# B&R Automation Studio project SortingStation
Automation Studio 4.12.4.107 SP; technology packages: mapp 5.23.1, mappCockpit 5.23.0, mappMotion 5.23.1, mappView 5.23.0

## Configuration Configuration

CPU X20CP1686X, AutomationRuntime H4.93, Build 4.1.2, Vc V4.73.0

### Task classes (Cpu.sw)
```
Cyclic#1:
  RSModelSor <- RSModelSort.prg
  ConveyorPr <- Source.Conveyor.ConveyorProgram.prg
  PuncherPro <- Source.Puncher.PuncherProgram.prg
Cyclic#2 (cycle 12000 us, tolerance 12000 us):
  MainMachin <- Source.MainMachine.MainMachineProgram.prg
  ColourSort <- Source.ColourSorter.ColourSorterProgram.prg
Cyclic#4:
  RecipesPro <- Source.Infrastructure.Recipes.RecipesProgram.prg
  Alarms <- Source.Infrastructure.Alarms.Alarms.prg
  HMIProgram <- Source.HMI.HMIProgram.prg
DataObjects: McAcpSys
NcDataObjects: McDriveLog
Binaries: TCLang, McAcpDrv, udbdef, McAcpSim, mvLoader, arflatprv, mCoWebSc, TCData, FWRules, arcoal, arsvcreg, OpcUaSrv, Settings, iomap, asfw, Role, ashwac, sysconf, AxisConfig, arconfig, AlarmsCore, AlarmsHist, TC, ashwd, User, Cam, Users
Libraries: McBase, MpAxis, McAxis, MpBase, McAcpAx, CoTrace, AsZip, FileIO, runtime, MpAlarmX, astime, standard, asstring, MpServer, MpFile, MpUserX, MpRecipe, sys_lib, asieccon, asbrstr, dataobj, asepl, asusb, aruser, arssl, powerlnk, arcert, ashw, aseth
```

### Hardware
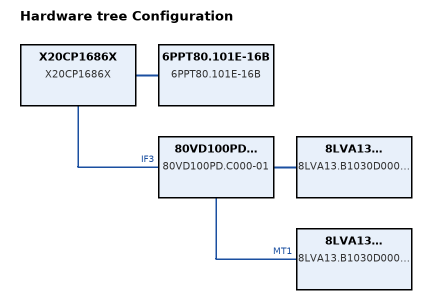
```
6PPT80.101E-16B : 6PPT80.101E-16B v1.0.6.0  [ETH1 -> X20CP1686X.IF2 [Cable Type=PowerlinkCable, Length=10, Version=1.0.0.3]]
  Terminal = true
  Startmode = 2
  Mode = Manual
  InternetAddress = 192.168.0.4
  Subnetmask = 255.255.255.0
  ScreenRotation = 180
  PasswordVNC = 
  SelectedFavoriteWeb = 192.168.0.3:81
  BrowserVKeyboard = 0
  PasswordCIFS = 
  PasswordService = 
80VD100PD.C000-01 : 80VD100PD.C000-01 v2.5.0.0  [PLK1 -> X20CP1686X.IF3 (NodeNumber=1) [Cable Type=PowerlinkCable, Length=10, Version=1.0.0.3]; MT2 -> 8LVA13.B1030D000-0.MT]
  DriveConfiguration/Module:
    McAcoposTypeID = AcoposMicroDConfig
    ActivateACOPOSSimulationOnPLC = 1
  DriveConfiguration/Channel[1]/RealAxis:
    AxisReference = gAxisConveyorMpLink
    MechanicalElementsIsInvisible = 0
  DriveConfiguration/Channel[1]/RealAxis/MechanicalElements/Gearbox:
    InputIsReadOnly = 0
    Input = 1
    OutputIsReadOnly = 0
    Output = 1
  DriveConfiguration/Channel[1]/RealAxis/MechanicalElements/RotaryToLinearTransformation:
    ReferenceDistanceIsReadOnly = 0
    ReferenceDistance = 1
  DriveConfiguration/Channel[1]/RealAxis/Controller:
    ModeIsReadOnly = 0
    Mode = PositionController
  DriveConfiguration/Channel[1]/RealAxis/Controller/Mode/Position:
    ProportionalGain = 50.0
    IntegrationTime = 0.0
    PredictionTime = 0.0004
    TotalDelayTime = 0.0004
  DriveConfiguration/Channel[1]/RealAxis/Controller/Mode/Speed:
    ProportionalGainIsReadOnly = 0
    ProportionalGain = 2.0
    IntegrationTimeIsReadOnly = 0
    IntegrationTime = 0.0
    FilterTimeIsReadOnly = 0
    FilterTime = 0.0
  DriveConfiguration/Channel[1]/RealAxis/Controller/Mode/LoopFilters:
    LoopFilterXIsReadOnly = 0
    LoopFilter1 = NotUsed
    LoopFilter2 = NotUsed
    LoopFilter3 = NotUsed
  DriveConfiguration/Channel[1]/RealAxis/Homing:
    ModeIsReadOnly = 0
    Mode = Direct
  DriveConfiguration/Channel[1]/RealAxis/Homing/Mode:
    Position = 0.0
    ReferencePulse = NotUsed
  DriveConfiguration/Channel[1]/RealAxis/Homing:
    RestorePositionVariable = 
  DriveConfiguration/Channel[1]/RealAxis/StopReaction:
    QuickstopIsReadOnly = 0
    Quickstop = DecelerationLimit
    DriveErrorIsReadOnly = 0
    DriveError = DecelerationLimit
  DriveConfiguration/Channel[1]/RealAxis/MovementErrorLimits:
    PositionError = 1.0
    VelocityErrorMonitoring = Automatic1
  DriveConfiguration/Channel[1]/RealAxis:
    JerkFilterIsReadOnly = 0
    JerkFilter = NotUsed
    ZeroVibrationFilter = NotUsed
  DriveConfiguration/Channel[1]/RealAxis/DigitalInputs/HomingSwitch:
    SourceIsReadOnly = 0
    Source = NotUsed
    Level = High
  DriveConfiguration/Channel[1]/RealAxis/DigitalInputs/PositiveLimitSwitch:
    SourceIsReadOnly = 0
    Source = NotUsed
    Level = High
  DriveConfiguration/Channel[1]/RealAxis/DigitalInputs/NegativeLimitSwitch:
    SourceIsReadOnly = 0
    Source = NotUsed
    Level = High
  DriveConfiguration/Channel[1]/RealAxis/DigitalInputs/Trigger1:
    Source = X2Trigger1
    Level = High
  DriveConfiguration/Channel[1]/RealAxis/DigitalInputs/Trigger2:
    Source = X2Trigger2
    Level = High
  DriveConfiguration/Channel[1]/RealAxis/DigitalInputs/Quickstop:
    Input = NotUsed
  DriveConfiguration/Channel[1]/RealAxis/Simulation:
    SimulationModeOnPLC = SetValueGeneration
    SimulationModeOnACOPOS = NotUsed
  DriveConfiguration/Channel[2]/RealAxis:
    AxisReference = gAxisPuncherMpLink
    MechanicalElementsIsInvisible = 0
  DriveConfiguration/Channel[2]/RealAxis/MechanicalElements/Gearbox:
    InputIsReadOnly = 0
    Input = 1
    OutputIsReadOnly = 0
    Output = 1
  DriveConfiguration/Channel[2]/RealAxis/MechanicalElements/RotaryToLinearTransformation:
    ReferenceDistanceIsReadOnly = 0
    ReferenceDistance = 1
  DriveConfiguration/Channel[2]/RealAxis/Controller:
    ModeIsReadOnly = 0
    Mode = PositionController
  DriveConfiguration/Channel[2]/RealAxis/Controller/Mode/Position:
    ProportionalGain = 50.0
    IntegrationTime = 0.0
    PredictionTime = 0.0004
    TotalDelayTime = 0.0004
  DriveConfiguration/Channel[2]/RealAxis/Controller/Mode/Speed:
    ProportionalGainIsReadOnly = 0
    ProportionalGain = 2.0
    IntegrationTimeIsReadOnly = 0
    IntegrationTime = 0.0
    FilterTimeIsReadOnly = 0
    FilterTime = 0.0
  DriveConfiguration/Channel[2]/RealAxis/Controller/Mode/LoopFilters:
    LoopFilterXIsReadOnly = 0
    LoopFilter1 = NotUsed
    LoopFilter2 = NotUsed
    LoopFilter3 = NotUsed
  DriveConfiguration/Channel[2]/RealAxis/Homing:
    ModeIsReadOnly = 0
    Mode = Direct
  DriveConfiguration/Channel[2]/RealAxis/Homing/Mode:
    Position = 0.0
    ReferencePulse = NotUsed
  DriveConfiguration/Channel[2]/RealAxis/Homing:
    RestorePositionVariable = 
  DriveConfiguration/Channel[2]/RealAxis/StopReaction:
    QuickstopIsReadOnly = 0
    Quickstop = DecelerationLimit
    DriveErrorIsReadOnly = 0
    DriveError = DecelerationLimit
  DriveConfiguration/Channel[2]/RealAxis/MovementErrorLimits:
    PositionError = 1.0
    VelocityErrorMonitoring = Automatic1
  DriveConfiguration/Channel[2]/RealAxis:
    JerkFilterIsReadOnly = 0
    JerkFilter = NotUsed
    ZeroVibrationFilter = NotUsed
  DriveConfiguration/Channel[2]/RealAxis/DigitalInputs/HomingSwitch:
    SourceIsReadOnly = 0
    Source = NotUsed
    Level = High
  DriveConfiguration/Channel[2]/RealAxis/DigitalInputs/PositiveLimitSwitch:
    SourceIsReadOnly = 0
    Source = NotUsed
    Level = High
  DriveConfiguration/Channel[2]/RealAxis/DigitalInputs/NegativeLimitSwitch:
    SourceIsReadOnly = 0
    Source = NotUsed
    Level = High
  DriveConfiguration/Channel[2]/RealAxis/DigitalInputs/Trigger1:
    Source = X2Trigger1
    Level = High
  DriveConfiguration/Channel[2]/RealAxis/DigitalInputs/Trigger2:
    Source = X2Trigger2
    Level = High
  DriveConfiguration/Channel[2]/RealAxis/DigitalInputs/Quickstop:
    Input = NotUsed
  DriveConfiguration/Channel[2]/RealAxis/Simulation:
    SimulationModeOnPLC = SetValueGeneration
    SimulationModeOnACOPOS = NotUsed
  DriveConfiguration/Channel[2]/RealAxis/AxisFeatures:
    FeatureRef[1] = CamAutomat
8LVA13.B1030D000-0 : 8LVA13.B1030D000-0 v2.2.0.3  [MT -> 80VD100PD.C000-01.MT2]
  M1/MotorParameters:
    MOTOR_AMB_TEMP_RATED = 40
8LVA13.B1030D000-0a : 8LVA13.B1030D000-0 v2.2.0.3  [MT -> 80VD100PD.C000-01.MT1]
  M1/MotorParameters:
    MOTOR_AMB_TEMP_RATED = 40
X20CP1686X : X20CP1686X v1.8.0.0
  Connector IF2:
    ActivateDevice = 1
    Mode = Manual
    InternetAddress = 192.168.0.3
    SubnetMask = 255.255.255.0
    ActivateSnmp = 2
  ConfigurationID = SortingStation_Configuration
  VolatileGlobalPvSize = 125535
  TimerDeviceType = EPLX2X
  TimerDevice = X20CP1686X.IF3
  Cyclic1Tolerance = 0
  Cyclic2Duration = 12000
  Cyclic2Tolerance = 12000
  FileDevice1
  FileDeviceName1 = RECIPES
  FileDevicePath1 = USER_PATH\recipes
  FtpUser1
  FtpUsername1 = admin
  FtpUserPassword1 = hWQDzdDXjPZQ9N0GtnGX4GsrlK/JakopLOxsvgAIz6U=
  FtpUserSalt1 = DV/Yji4l
  FTPAccessRight1 = 0
  FTPdevice1 = ALL
  ActivateOpcUa = 1
  OpcUaInformationModels_PV_Version = 2
  OpcUaInformationModel_Facet = 0
  OpcUaInformationModel_TypeInformation = 0
  OpcUaInformationModel_BaseObjectTypeForStructures = 0
```

- Physical/Configuration/X20CP1686X/IoMap.iom: same as Physical/Configuration/X20CP1686X/Cpu.per
### AxisConfig.axis - X20CP1686X/mappMotion/AxisConfig.axis
```
Element gAxisConveyorMpLink (Type=axis)
  BaseTypeIsReadOnly = 0
  BaseType = LinearPeriodic
    MeasurementUnit = 5066068
    MeasurementResolutionIsReadOnly = 0
    MeasurementResolution = 0.01
    CountDirectionIsReadOnly = 0
    CountDirection = Standard
    PeriodSettings:
      Period = 580
  MovementLimitsIsReadOnly = 0
  MovementLimits = Internal
    Position:
      LowerLimitMin = -1.79769313486231E308
      UpperLimitMax = 1.79769313486231E308
      LowerLimit = -1000.0
      UpperLimit = 1000.0
    VelocityIsReadOnly = 0
    Velocity:
      VelocityMax = 3.4E38
      Velocity = 500
    AccelerationIsReadOnly = 0
    Acceleration:
      AccelerationMax = 3.4E38
      Acceleration = 5000
    DecelerationIsReadOnly = 0
    Deceleration:
      DecelerationMax = 3.4E38
      Deceleration = 5000
  Alarms = MpAlarmX
    mapp.AlarmX.Core.Configuration:
      [2]:
        Severity = 0
Element gAxisPuncherMpLink (Type=axis)
  BaseTypeIsReadOnly = 0
  BaseType = Linear
    MeasurementUnit = 5066068
    MeasurementResolutionIsReadOnly = 0
    MeasurementResolution = 0.01
    CountDirectionIsReadOnly = 0
    CountDirection = Standard
  MovementLimitsIsReadOnly = 0
  MovementLimits = Internal
    Position:
      LowerLimitMin = -1.79769313486231E308
      UpperLimitMax = 1.79769313486231E308
      LowerLimit = 0
      UpperLimit = 0.46
    VelocityIsReadOnly = 0
    Velocity:
      VelocityMax = 3.4E38
      Velocity = 100000
    AccelerationIsReadOnly = 0
    Acceleration:
      AccelerationMax = 3.4E38
      Acceleration = 200000
    DecelerationIsReadOnly = 0
    Deceleration:
      DecelerationMax = 3.4E38
      Deceleration = 200000
  Alarms = MpAlarmX
    mapp.AlarmX.Core.Configuration:
      [2]:
        Severity = 0
```

### Cam.axisfeature - X20CP1686X/mappMotion/Cam.axisfeature
```
Element CamAutomat (Type=axisfeature)
  Type = CamAutomat
    CamAutomatType = ACOPOS
      CommonParameters:
        Master:
          ValueSource = SetPosition
            AxisReference = gAxisConveyorMpLink
            MaxVelocity = 500
          StartPosition = 0.0
          StartInterval = MasterAxisPeriod
        AdvancedParameters:
          StartStateParameters:
            StartState = 0
            RelMasterStartPos = 0.0
          AdditiveAxes:
            AdditiveMasterValueSource = NotUsed
            AdditiveSlaveValueSource = NotUsed
          MasterStartPositionMode = NotEvaluatedAnew
          ControlSettings:
            CrossLeftBoundary = PositionLimitedHorizontal
            CamChangeImmediately = CurrentMasterMoveDir
          MessageSettings:
            ErrorsInStandby = NoErrorMessages
          TriggerAndLatch:
            Trigger1Delay = 0.0
            Trigger2Delay = 0.0
            SlaveLatchParID = 0
          EventParIDs
          StartIntervals
          Factors:
            SlaveFactorParID = 0
      States:
        State0 = Used
          Events:
            Event[0]:
              Type = Signal1FromPLC
              Transition = Immediately
              SynchronousUpdate = NotUsed
              NextState = 1
        State[1]:
          Cam = Predefined
            PredefinedCam = OneToOne
          MasterFactor = 20000
          SlaveFactor = 20000
          CompensationMode = DistancesBetweenExitEntryPoints
            MasterDistance = 100
            SlaveDistance = 20
            AdvancedParameters = NotUsed
          AdvancedParameters:
            RepeatCounterInit = 0
            MasterValueSource = CommonMaster
          Events:
            Event[0]:
              Type = StateEnd
              Transition = Immediately
              SynchronousUpdate = NotUsed
              NextState = 2
        State[2]:
          Cam = Predefined
            PredefinedCam = ZeroPoint
          MasterFactor = 1
          SlaveFactor = 0
          CompensationMode = DistancesBetweenExitEntryPoints
            MasterDistance = 100
            SlaveDistance = -220
            AdvancedParameters = NotUsed
          AdvancedParameters:
            RepeatCounterInit = 0
            MasterValueSource = CommonMaster
          Events:
            Event[0]:
              Type = StateEnd
              Transition = Immediately
              SynchronousUpdate = NotUsed
              NextState = 0
```

- Safety project (password-protected, skipped)

### AlarmsCore.mpalarmxcore - X20CP1686X/mappServices/AlarmsCore.mpalarmxcore
```
Element gAlarmXCoreMpLink (Type=mpalarmxcore)
  mapp.AlarmX.Core:
    Mapping:
      [0]
    BySeverity:
      [0]:
        Severity = 1
        [0] = Reaction
          Name = STOP
      [1]:
        Severity = 2
        [0] = Reaction
          Name = STOP_ON_PHASE
  mapp.AlarmX.Core.Configuration:
    [0]:
      Name = ColourSorterTimeoutSetLanes
      Message = {$Source/ColourSorter/Alarms/ColourSorterTimeoutSetLanes}
    [1]:
      Name = ColourSorterMissingCap
      Message = {$Source/ColourSorter/Alarms/ColourSorterMissingCap}
    [2]:
      Name = ColourSorterInvalidSensorsCombinationLane1
      Message = {$Source/ColourSorter/Alarms/ColourSorterInvalidSensorsCombinationLane1}
      Behavior = PersistentAlarm
    [3]:
      Name = ColourSorterInvalidSensorsCombinationLane2
      Message = {$Source/ColourSorter/Alarms/ColourSorterInvalidSensorsCombinationLane2}
      Behavior = PersistentAlarm
    [4]:
      Name = ColourSorterInvalidParametersCombination
      Message = {$Source/ColourSorter/Alarms/ColourSorterInvalidParametersCombination}
      Behavior = PersistentAlarm
    [5]:
      Name = ColourSorterFullLanes
      Message = {$Source/ColourSorter/Alarms/ColourSorterFullLanes}
      Behavior = PersistentAlarm
    [6]:
      Name = ConveyorTimeoutHoming
      Message = {$Source/Conveyor/Alarms/ConveyorTimeoutHoming}
    [7]:
      Name = ConveyorTimeoutPowerOn
      Message = {$Source/Conveyor/Alarms/ConveyorTimeoutPowerOn}
    [8]:
      Name = ConveyorAxisError
      Message = {$Source/Conveyor/Alarms/ConveyorAxisError}
      Behavior = PersistentAlarm
    [9]:
      Name = ConveyorInitFail
      Message = {$Source/Conveyor/Alarms/ConveyorInitFail}
    [10]:
      Name = ConveyorTooManyCaps
      Message = {$Source/Conveyor/Alarms/ConveyorTooManyCaps}
      Behavior = PersistentAlarm
    [11]:
      Name = PuncherAxisError
      Message = {$Source/Puncher/Alarms/PuncherAxisError}
      Behavior = PersistentAlarm
    [12]:
      Name = PuncherInvalidSensorsCombination
      Message = {$Source/Puncher/Alarms/PuncherInvalidSensorsCombination}
      Behavior = PersistentAlarm
    [13]:
      Name = PuncherTimeoutHoming
      Message = {$Source/Puncher/Alarms/PuncherTimeoutHoming}
    [14]:
      Name = PuncherTimeoutPowerOn
      Message = {$Source/Puncher/Alarms/PuncherTimeoutPowerOn}
    [15]:
      Name = PuncherTimeoutPunchBackward
      Message = {$Source/Puncher/Alarms/PuncherTimeoutPunchBackward}
    [16]:
      Name = PuncherTimeoutPunchForward
      Message = {$Source/Puncher/Alarms/PuncherTimeoutPunchForward}
    [17]:
      Name = PuncherAxisTimeout
      Message = {$Source/Puncher/Alarms/PuncherAxisTimeout}
    [18]:
      Name = MainMachineEmergencyCircuitInterrupted
      Message = {$Source/MainMachine/Alarms/MainMachineEmergencyCircuitInterrupted}
      Behavior = PersistentAlarm
    [19]:
      Name = MainMachineCommunicationLost
      Message = {$Source/MainMachine/Alarms/MainMachineCommunicationLost}
      Severity = 2
      Behavior = PersistentAlarm
    [20]:
      Name = MainMachineInitializationTimeout
      Message = {$Source/MainMachine/Alarms/MainMachineInitializationTimeout}
    [21]:
      Name = MainMachinePickingStationInError
      Message = {$Source/MainMachine/Alarms/MainMachinePickingStationInError}
      Severity = 2
      Behavior:
        MultipleInstances = FALSE
    [22]:
      Name = MainMachinePickingStationNotInLinkMode
      Message = {$Source/MainMachine/Alarms/MainMachinePickingStationNotInLinkMode}
      Behavior = PersistentAlarm
    [23]:
      Name = MainMachineCapMissing
      Message = {$Source/MainMachine/Alarms/MainMachineCapMissing}
```

### AlarmsHist.mpalarmxhistory - X20CP1686X/mappServices/AlarmsHist.mpalarmxhistory
```
Element gAlarmXHistoryMpLink (Type=mpalarmxhistory)
```

### Recipes.mprecipexml - X20CP1686X/mappServices/Recipes.mprecipexml
```
Element gRecipesXmlMpLink (Type=mprecipexml)
  Alarms = MpAlarmX
```

### Users.mpuserx - X20CP1686X/mappServices/Users.mpuserx
```
Element UserMgmtX (Type=mpuserx)
  Mgr:
    LoginAttempts = 0
  ServerSettings:
    Server:
      AdditionalUserData:
        [0] = mail
        [1] = telephoneNumber
  Users:
    DefUser#1:
      id = admin
      name = Andrea Pennisi
      lang = it
      unit = imperial
    DefUser#2:
      id = Anonymous
      lang = en
      unit = metric
  Groups:
    DefGroup#1:
      id = Everyone
      level = 0
    DefGroup#2:
      id = Administrators
      admin = TRUE
```

## Logical view

Binary libraries used (declarations not repeated): operator, runtime, astime, AsIecCon, McBase 5.23.1, MpAxis 5.23.1, McAxis 5.23.1, MpBase 5.23.0, McAcpAx 5.23.1, CoTrace 5.23.0, AsZip, FileIO, MpAlarmX 5.23.1, standard, asstring, MpServer 5.23.0, MpFile 5.23.1, MpUserX 5.23.1, MpRecipe 5.23.1, sys_lib


### Program Logical/RSModelSort (IEC) - IO Interface to the RobotStudio model (Sort IOs)

#### Main.st - Init, cyclic, exit code
```iecst
PROGRAM _INIT
	diCapOnSortingConveyor;
	diHolePuncherForward;
	diHolePuncherBack;
	diColourDetection;
	diCapColourNotBlack;
	diCapColourMetallic;
	diLaneGate1Forward;
	diLaneGate1Back;
	diLaneGate2Forward;
	diLaneGate2Back;
	diLaneTop;
	aiPuncherAxisActPos;
	doHolePuncher;
	doSortingConveyorClear;
	doCapStopper;
	doLaneGate1;
	doLaneGate2;
	aoSortingConveyorSetSpeed;
	aoPuncherAxisSetPos;
	doLaneStopper1Clear;
	doLaneStopper2Clear;
	doLaneStopper3Clear;
	doCreateCapForSorting;
END_PROGRAM

PROGRAM _CYCLIC

	// Colour sorter
	gColourSorter.Interface.Inputs.CapAtStartPosition := diColourDetection;
	gColourSorter.Interface.Inputs.CapAtExitPosition := diLaneTop;
	gColourSorter.Interface.Inputs.ColourIsMetallic := diCapColourMetallic;
	gColourSorter.Interface.Inputs.ColourIsNotBlack := diCapColourNotBlack;
	gColourSorter.Interface.Inputs.Lane1GateBackward := diLaneGate1Back;
	gColourSorter.Interface.Inputs.Lane1GateForward := diLaneGate1Forward;
	gColourSorter.Interface.Inputs.Lane2GateBackward := diLaneGate2Back;
	gColourSorter.Interface.Inputs.Lane2GateForward := diLaneGate2Forward;

	doLaneGate1 := gColourSorter.Interface.Outputs.Lane1GateForward;
	doLaneGate2 := gColourSorter.Interface.Outputs.Lane2GateForward;
	doCapStopper := gColourSorter.Interface.Outputs.StopperForward;

	// Conveyor
	gConveyor.Interface.Inputs.CapInStartPosition := diCapOnSortingConveyor;

	aoSortingConveyorSetSpeed := gConveyor.Interface.Outputs.SetSpeed/1000;

	// Puncher
	gPuncher.Interface.Inputs.ActualPosition := aiPuncherAxisActPos*1000;
	gPuncher.Interface.Inputs.PunchIsForward := diHolePuncherForward;
	gPuncher.Interface.Inputs.PunchIsBackward := diHolePuncherBack;

	aoPuncherAxisSetPos := LREAL_TO_REAL(gPuncher.Interface.Outputs.SetPosition/1000);
	doHolePuncher := gPuncher.Interface.Outputs.PunchForward;

END_PROGRAM

PROGRAM _EXIT
	(* Insert code here *)

END_PROGRAM
```

#### Variables.var - Local variables
```iecst
(*Inputs*)
VAR
	diCapOnSortingConveyor : BOOL := 0;
	diHolePuncherForward : BOOL := 0;
	diHolePuncherBack : BOOL := 0;
	diColourDetection : BOOL := 0;
	diCapColourNotBlack : BOOL := 0;
	diCapColourMetallic : BOOL := 0;
	diLaneGate1Forward : BOOL := 0;
	diLaneGate1Back : BOOL := 0;
	diLaneGate2Forward : BOOL := 0;
	diLaneGate2Back : BOOL := 0;
	diLaneTop : BOOL := 0;
	aiPuncherAxisActPos : REAL := 0.0; (*[m]*)
END_VAR
(*Outputs*)
VAR
	doHolePuncher : BOOL := 0;
	doSortingConveyorClear : BOOL := 0;
	doCapStopper : BOOL := 0;
	doLaneGate1 : BOOL := 0;
	doLaneGate2 : BOOL := 0;
	aoSortingConveyorSetSpeed : REAL := 0.0; (*[m/s]*)
	aoPuncherAxisSetPos : REAL := 0.0; (*[m]*)
END_VAR
(*Model Interaction*)
VAR
	doLaneStopper1Clear : BOOL := 0;
	doLaneStopper2Clear : BOOL := 0;
	doLaneStopper3Clear : BOOL := 0;
	doCreateCapForSorting : BOOL := 0;
END_VAR
```

### AlarmsGlobalVariables.var
```iecst
VAR
	gAlarms : AlarmsType;
END_VAR
```

### AlarmsGlobalTypes.typ
```iecst
TYPE
	AlarmsType : 	STRUCT
		Feedbacks : AlarmsFeedbacksType;
		MpAlarmXListUIConnect : MpAlarmXListUIConnectType;
	END_STRUCT;
	AlarmsFeedbacksType : 	STRUCT
		Pendings : UDINT;
	END_STRUCT;
END_TYPE
```

### Program Logical/Source/Infrastructure/Alarms/Alarms (IEC)

#### Main.st - Init, cyclic, exit code
```iecst
PROGRAM _INIT
	// This program is used to manage the machine alarms. Alarms are set/reset in the modules.

	MpAlarmXCoreFB(MpLink := ADR(gAlarmXCoreMpLink), Enable := TRUE);

	MpAlarmXHistoryFB(MpLink := ADR(gAlarmXHistoryMpLink), Enable := TRUE, DeviceName := ADR('ALARMS'));

	MpAlarmXListUIFB(MpLink :=  ADR(gAlarmXCoreMpLink), Enable := TRUE, UIConnect := ADR(gAlarms.MpAlarmXListUIConnect));

END_PROGRAM

PROGRAM _CYCLIC
	MpAlarmXCoreFB();

	MpAlarmXHistoryFB();

	MpAlarmXListUIFB();

	gAlarms.Feedbacks.Pendings := MpAlarmXCoreFB.PendingAlarms;

END_PROGRAM

PROGRAM _EXIT
	MpAlarmXCoreFB.Enable := FALSE;
	MpAlarmXCoreFB();

	MpAlarmXHistoryFB.Enable := FALSE;
	MpAlarmXHistoryFB();

	MpAlarmXListUIFB.Enable := FALSE;
	MpAlarmXListUIFB();

END_PROGRAM
```

#### Variables.var - Local variables
```iecst
VAR
	MpAlarmXCoreFB : MpAlarmXCore;
	MpAlarmXHistoryFB : MpAlarmXHistory;
	MpAlarmXListUIFB : MpAlarmXListUI;
END_VAR
```

### RecipesGlobalVariables.var
```iecst
VAR
	gRecipes : MpRecipeUIConnectType;
END_VAR
```

### Program Logical/Source/Infrastructure/Recipes/RecipesProgram (IEC)

#### Main.st - Init, cyclic, exit code
```iecst
PROGRAM _INIT

	MpRecipeXmlFB(MpLink := ADR(gRecipesXmlMpLink), Enable := TRUE, DeviceName := ADR('RECIPES'));
	MpRecipeUIFB(MpLink := ADR(gRecipesXmlMpLink), Enable := TRUE, UIConnect := ADR(gRecipes));

	gRecipes.New.FileName := 'Default.xml';
END_PROGRAM

PROGRAM _CYCLIC
	MpRecipeXmlFB(ErrorReset := gMainMachine.Commands.Reset AND MpRecipeXmlFB.Error);
	MpRecipeUIFB(ErrorReset := gMainMachine.Commands.Reset AND MpRecipeUIFB.Error);

	// Manage the recipe change
	IF MpRecipeXmlFB.StatusID = ERR_OK AND MpRecipeUIFB.StatusID = ERR_OK THEN
		gRecipes.Recipe.List.SelectedIndex := MIN(gRecipes.Recipe.List.SelectedIndex,gRecipes.Recipe.List.MaxSelection);
		// Load recipe on power on of plc or if a new recipe is selected from HMI
		IF NOT InitDone OR gRecipes.Recipe.List.SelectedIndex <> LastRecipeIndex THEN
			gRecipes.Recipe.Load := TRUE;
			InitDone := TRUE;
			LastRecipeIndex := gRecipes.Recipe.List.SelectedIndex;
		END_IF
		gRecipes.Recipe.Delete := FALSE;
		gRecipes.Recipe.Save := FALSE;
		IF gRecipes.New.Create THEN
			gRecipes.New.Create := FALSE;
			gRecipes.New.FileName := 'Default.xml';
		END_IF
	END_IF

END_PROGRAM

PROGRAM _EXIT
	MpRecipeXmlFB.Enable := FALSE;
	MpRecipeXmlFB();

	MpRecipeUIFB.Enable := FALSE;
	MpRecipeUIFB();
END_PROGRAM
```

#### Variables.var - Local variables
```iecst
VAR
	MpRecipeXmlFB : MpRecipeXml;
	MpRecipeUIFB : MpRecipeUI;
	InitDone : BOOL;
	LastRecipeIndex : UINT;
END_VAR
```

### ColourSorterGlobalTypes.typ
```iecst
TYPE
	ColourSorterType : 	STRUCT  (*ColourSorter Main type*)
		Commands : ColourSorterCommadsType;
		Feedbacks : ColourSorterFeedbacksType;
		Interface : ColourSorterInterfaceType;
		Parameters : ColourSorterParametersType;
	END_STRUCT;
	ColourSorterCommadsType : 	STRUCT  (*ColourSorter Commands type*)
		Enable : BOOL;
		Reset : BOOL;
		Manual : ColourSorterManualCommadsType;
		Automatic : ColourSorterAutomaticCommadsType;
	END_STRUCT;
	ColourSorterFeedbacksType : 	STRUCT  (*ColourSorter Feedbacks type*)
		Enabled : BOOL;
		WaitingCap : BOOL;
		Error : BOOL;
		WaitingStart : BOOL;
		CapSorted : BOOL;
		InitDone : BOOL;
		InitPosition : BOOL;
	END_STRUCT;
	ColourSorterInterfaceType : 	STRUCT  (*ColourSorter Interface type*)
		Inputs : ColourSorterInterfaceInputsType;
		Outputs : ColourSorterInterfaceOutputsType;
	END_STRUCT;
	ColourSorterInterfaceOutputsType : 	STRUCT  (*ColourSorter Interface Output type*)
		StopperForward : BOOL;
		Lane1GateForward : BOOL;
		Lane2GateForward : BOOL;
	END_STRUCT;
	ColourSorterInterfaceInputsType : 	STRUCT  (*ColourSorter Interface Input type*)
		CapAtStartPosition : BOOL;
		ColourIsNotBlack : BOOL;
		ColourIsMetallic : BOOL;
		Lane1GateBackward : BOOL;
		Lane1GateForward : BOOL;
		Lane2GateBackward : BOOL;
		Lane2GateForward : BOOL;
		CapAtExitPosition : BOOL;
	END_STRUCT;
	ColourSorterAutomaticCommadsType : 	STRUCT  (*ColourSorter Commands type*)
		Init : BOOL;
		Start : BOOL;
	END_STRUCT;
	ColourSorterManualCommadsType : 	STRUCT  (*ColourSorter Commands type*)
		Enable : BOOL;
		Lane1Forward : BOOL;
		Lane2Forward : BOOL;
		StopperForward : BOOL;
	END_STRUCT;
	ColourSorterParametersType : 	STRUCT  (*ColourSorter Commands type*)
		GreyLane : USINT := 3;
		RedLane : USINT := 1;
		BlackLane : USINT := 2;
	END_STRUCT;
END_TYPE
```

### ColourSorterGlobalVariables.var
```iecst
VAR
	gColourSorter : ColourSorterType;
END_VAR
```

### Program Logical/Source/ColourSorter/ColourSorterProgram (IEC)

#### Main.st - Init, cyclic, exit code
```iecst
//******************************************************************************************************
// Program: 	ColourSorterProgram
// Author: 		Andrea Pennisi
// Rev.: 		1.0.0
// Date:		5.12.2023
//
// Description:
// This module is used to sort the caps by color.
// Only pneumatic motion in this module. mappRecipesX is used to manage the lanes order.
//******************************************************************************************************

PROGRAM _INIT

    ResetOutputsAction;
    ResetFeedbacksAction;

	MpRecipeRegParFB(MpLink := ADR(gRecipesXmlMpLink), Enable := TRUE, PVName := ADR('gColourSorter.Parameters'));

    MachineState.NextState := WAITING_INIT;

END_PROGRAM

PROGRAM _CYCLIC
    // Recipe
	MpRecipeRegParFB(ErrorReset := gColourSorter.Commands.Reset AND MpRecipeRegParFB.Error);

    // Enable module
    IF NOT gColourSorter.Commands.Enable THEN
        ResetOutputsAction;
		ResetFeedbacksAction;
		ResetAlarmsAction;
        RETURN;
    END_IF

	IF EDGENEG(gColourSorter.Commands.Automatic.Start) THEN
		IF MachineState.NextState <> ERROR THEN
			MachineState.NextState := WAITING_START;
		END_IF
	END_IF

	IF EDGEPOS(gColourSorter.Commands.Automatic.Init) THEN
		IF MachineState.NextState <> ERROR THEN
			MachineState.NextState := WAITING_INIT;
		END_IF
	END_IF

	// Alarms
	SetAlarmsAction;

    // Machine state
    MachineStateManagementAction;
    CASE MachineState.ActualState OF

		WAITING_INIT:
			MachineState.TimeoutTimer.PT := T#0S; // Timeout disabled in this state
			IF MachineState.NewTriggerState THEN
				ResetOutputsAction;
				gColourSorter.Feedbacks.CapSorted := FALSE;
			END_IF

			IF gColourSorter.Commands.Automatic.Init THEN
				Internal.Lane1ForwardPositionRequest := FALSE;
				Internal.Lane2ForwardPositionRequest := FALSE;
				Internal.CapOnProcess := FALSE;
				gColourSorter.Feedbacks.CapSorted := FALSE;

				MachineState.NextState := SET_LANES;

			ELSIF gColourSorter.Commands.Manual.Enable THEN
				MachineState.NextState := MANUALS;

			END_IF

		MANUALS:
			MachineState.TimeoutTimer.PT := T#0S; // Timeout disabled in this state
			// Manual commands
			gColourSorter.Interface.Outputs.Lane1GateForward := gColourSorter.Commands.Manual.Lane1Forward;
			gColourSorter.Interface.Outputs.Lane2GateForward := gColourSorter.Commands.Manual.Lane2Forward;
			gColourSorter.Interface.Outputs.StopperForward := gColourSorter.Commands.Manual.StopperForward;

			IF NOT gColourSorter.Commands.Manual.Enable THEN
				MachineState.NextState := WAITING_INIT;
			END_IF

		SET_LANES:
			MachineState.TimeoutTimer.PT := T#3S;
			IF MachineState.NewTriggerState THEN
				Internal.Lane1PositionOk := FALSE;
				Internal.Lane2PositionOk := FALSE;
			END_IF

			gColourSorter.Interface.Outputs.Lane1GateForward := Internal.Lane1ForwardPositionRequest;
			gColourSorter.Interface.Outputs.Lane2GateForward := Internal.Lane2ForwardPositionRequest;

			IF Internal.Lane1ForwardPositionRequest THEN
				Internal.Lane1PositionOk := gColourSorter.Interface.Inputs.Lane1GateForward;
			ELSE
				Internal.Lane1PositionOk := gColourSorter.Interface.Inputs.Lane1GateBackward;
			END_IF

			IF Internal.Lane2ForwardPositionRequest THEN
				Internal.Lane2PositionOk := gColourSorter.Interface.Inputs.Lane2GateForward;
			ELSE
				Internal.Lane2PositionOk := gColourSorter.Interface.Inputs.Lane2GateBackward;
			END_IF

			IF Internal.Lane1PositionOk AND Internal.Lane2PositionOk THEN
				IF Internal.CapOnProcess THEN
					MachineState.NextState := STOPPER_BACKWARD;
				ELSE
					MachineState.NextState := STOPPER_FORWARD;
				END_IF
			END_IF

		STOPPER_FORWARD:
			MachineState.TimeoutTimer.PT := T#10S;
			gColourSorter.Interface.Outputs.StopperForward := TRUE;
			IF MachineState.TimeoutTimer.ET > T#250MS THEN
				MachineState.NextState := WAITING_START;
			END_IF

		WAITING_START:
			MachineState.TimeoutTimer.PT := T#0S; // Timeout disabled in this state

			IF gColourSorter.Commands.Automatic.Start THEN
				MachineState.NextState := WAITING_CAP;

			ELSIF gColourSorter.Commands.Manual.Enable THEN
				MachineState.NextState := MANUALS;
			END_IF

        WAITING_CAP:
			MachineState.TimeoutTimer.PT := T#0S; // Timeout disabled in this state
			IF MachineState.NewTriggerState THEN
				Internal.CapOnProcess := FALSE;
			END_IF

			IF gColourSorter.Interface.Inputs.CapAtStartPosition THEN
				Internal.CapOnProcess := TRUE;
				gColourSorter.Feedbacks.CapSorted := FALSE;
                MachineState.NextState := DETECTING_COLOR;
            END_IF

		DETECTING_COLOR:
			MachineState.TimeoutTimer.PT := T#10S;
			IF gColourSorter.Interface.Inputs.ColourIsMetallic THEN
				// GRAY
				Internal.Lane1ForwardPositionRequest := (gColourSorter.Parameters.GreyLane = 1);
				Internal.Lane2ForwardPositionRequest := (gColourSorter.Parameters.GreyLane = 2);

			ELSIF gColourSorter.Interface.Inputs.ColourIsNotBlack THEN
				// RED
				Internal.Lane1ForwardPositionRequest := (gColourSorter.Parameters.RedLane = 1);
				Internal.Lane2ForwardPositionRequest := (gColourSorter.Parameters.RedLane = 2);

			ELSE
				// BLACK
				Internal.Lane1ForwardPositionRequest := (gColourSorter.Parameters.BlackLane = 1);
				Internal.Lane2ForwardPositionRequest := (gColourSorter.Parameters.BlackLane = 2);

			END_IF

			IF MachineState.TimeoutTimer.ET > T#250MS THEN
				MachineState.NextState := SET_LANES;
			END_IF

		STOPPER_BACKWARD:
			MachineState.TimeoutTimer.PT := T#0S; // Timeout disabled in this state

			gColourSorter.Interface.Outputs.StopperForward := FALSE;

			MachineState.NextState := WAITING_CAP_EXIT;

		WAITING_CAP_EXIT:
			MachineState.TimeoutTimer.PT := T#15S;

			IF gColourSorter.Interface.Inputs.CapAtExitPosition THEN
				gColourSorter.Feedbacks.CapSorted := TRUE;
				MachineState.NextState := STOPPER_FORWARD;
			END_IF

		ERROR:
			MachineState.TimeoutTimer.PT := T#0S; // Timeout disabled in this state
			ResetOutputsAction;
			IF NOT Internal.Error THEN
				MachineState.NextState := WAITING_INIT;
			END_IF

        ELSE
            MachineState.NextState := WAITING_INIT;

    END_CASE

    FeedbacksUpdateAction;

END_PROGRAM

PROGRAM _EXIT
	MpRecipeRegParFB(Enable := FALSE);

END_PROGRAM
```

#### Types.typ - Local data types
```iecst
TYPE
	MachineStateType : 	STRUCT  (*Machine state main type*)
		OldState : MachineStateEnum; (*Actual state*)
		ActualState : MachineStateEnum; (*Actual state*)
		NextState : MachineStateEnum; (*Next state*)
		NewTriggerState : BOOL; (*Trigger state change*)
		TimeoutTimer : TON; (*State timeout*)
	END_STRUCT;
	MachineStateEnum :
		( (*Machine State enumeration*)
		WAITING_INIT,
		MANUALS,
		WAITING_START,
		STOPPER_FORWARD, (*INIT state*)
		SET_LANES, (*WAITING state*)
		WAITING_CAP, (*ERROR state*)
		DETECTING_COLOR,
		STOPPER_BACKWARD,
		WAITING_CAP_EXIT,
		ERROR
		);
	InternalType : 	STRUCT
		Error : BOOL;
		Lane1ForwardPositionRequest : BOOL;
		Lane2ForwardPositionRequest : BOOL;
		Lane1PositionOk : BOOL;
		Lane2PositionOk : BOOL;
		CapOnProcess : BOOL;
		LaneFullTimeout : TON := (PT:=T#10S);
	END_STRUCT;
END_TYPE
```

#### Variables.var - Local variables
```iecst
VAR
	MachineState : MachineStateType;
	Internal : InternalType;
	MpRecipeRegParFB : MpRecipeRegPar; (*Recipe register functionblock*)
END_VAR
```

#### Actions.st
```iecst
ACTION FeedbacksUpdateAction:

	gColourSorter.Feedbacks.Enabled := TRUE;
    gColourSorter.Feedbacks.WaitingCap := MachineState.ActualState = WAITING_CAP;
    gColourSorter.Feedbacks.Error := MachineState.ActualState = ERROR;
	gColourSorter.Feedbacks.InitPosition := gColourSorter.Interface.Inputs.Lane1GateBackward AND gColourSorter.Interface.Inputs.Lane2GateBackward;
	gColourSorter.Feedbacks.InitDone := gColourSorter.Feedbacks.InitPosition AND gColourSorter.Commands.Automatic.Init;

END_ACTION

ACTION ResetOutputsAction:

    memset(ADR(gColourSorter.Interface.Outputs),0,SIZEOF(gColourSorter.Interface.Outputs));

END_ACTION

ACTION ResetFeedbacksAction:

    memset(ADR(gColourSorter.Feedbacks),0,SIZEOF(gColourSorter.Feedbacks));

END_ACTION

ACTION MachineStateManagementAction:

    // Machine state timeout check
    MachineState.TimeoutTimer(IN := MachineState.TimeoutTimer.PT <> T#0S AND NOT MachineState.NewTriggerState);

	// Machine state change state logic
	MachineState.NewTriggerState := (MachineState.ActualState <> MachineState.NextState);
	IF MachineState.NewTriggerState THEN
		MachineState.OldState := MachineState.ActualState;
	END_IF
	MachineState.ActualState := MachineState.NextState;

END_ACTION

ACTION SetAlarmsAction:

	IF gColourSorter.Commands.Reset THEN
		Internal.Error := FALSE;
	END_IF

	// Timeouts alarms
	IF MachineState.TimeoutTimer.Q THEN
		CASE MachineState.ActualState OF
			SET_LANES: MpAlarmXSet(gAlarmXCoreMpLink,'ColourSorterTimeoutSetLanes'); // Edge alarm!
			WAITING_CAP_EXIT: MpAlarmXSet(gAlarmXCoreMpLink,'ColourSorterMissingCap'); // Edge alarm!
		END_CASE
		Internal.Error := TRUE;
		MachineState.NextState := ERROR;
	END_IF

	// ColourSorterInvalidSensorsCombinationLane1
	IF gColourSorter.Interface.Inputs.Lane1GateBackward AND gColourSorter.Interface.Inputs.Lane1GateForward THEN
		MpAlarmXSet(gAlarmXCoreMpLink,'ColourSorterInvalidSensorsCombinationLane1'); // Periodic alarm!
		Internal.Error := TRUE;
		MachineState.NextState := ERROR;
	ELSE
		MpAlarmXReset(gAlarmXCoreMpLink,'ColourSorterInvalidSensorsCombinationLane1');
	END_IF

	// ColourSorterInvalidSensorsCombinationLane2
	IF gColourSorter.Interface.Inputs.Lane1GateBackward AND gColourSorter.Interface.Inputs.Lane1GateForward THEN
		MpAlarmXSet(gAlarmXCoreMpLink,'ColourSorterInvalidSensorsCombinationLane2'); // Periodic alarm!
		Internal.Error := TRUE;
		MachineState.NextState := ERROR;
	ELSE
		MpAlarmXReset(gAlarmXCoreMpLink,'ColourSorterInvalidSensorsCombinationLane2');
	END_IF

	// ColourSorterInvalidParametersCombination
	IF gColourSorter.Parameters.BlackLane < 1 OR gColourSorter.Parameters.BlackLane > 3
		OR gColourSorter.Parameters.GreyLane < 1 OR gColourSorter.Parameters.GreyLane > 3
		OR gColourSorter.Parameters.RedLane < 1 OR gColourSorter.Parameters.RedLane > 3
		OR gColourSorter.Parameters.BlackLane = gColourSorter.Parameters.RedLane
		OR gColourSorter.Parameters.BlackLane = gColourSorter.Parameters.GreyLane
		OR gColourSorter.Parameters.GreyLane = gColourSorter.Parameters.RedLane THEN

		MpAlarmXSet(gAlarmXCoreMpLink,'ColourSorterInvalidParametersCombination'); // Periodic alarm!
		Internal.Error := TRUE;
		MachineState.NextState := ERROR;
	ELSE
		MpAlarmXReset(gAlarmXCoreMpLink,'ColourSorterInvalidParametersCombination');
	END_IF

	// ColourSorterFullLanes
	Internal.LaneFullTimeout(IN:=gColourSorter.Interface.Inputs.CapAtExitPosition);
	IF Internal.LaneFullTimeout.Q THEN
		Internal.Error := TRUE;
		MachineState.NextState := ERROR;
		MpAlarmXSet(gAlarmXCoreMpLink,'ColourSorterFullLanes'); // Periodic alarm!
	ELSE
		MpAlarmXReset(gAlarmXCoreMpLink,'ColourSorterFullLanes');
	END_IF

END_ACTION

ACTION ResetAlarmsAction:

	MpAlarmXReset(gAlarmXCoreMpLink,'ColourSorterInvalidSensorsCombinationLane1');
	MpAlarmXReset(gAlarmXCoreMpLink,'ColourSorterInvalidSensorsCombinationLane2');
	MpAlarmXReset(gAlarmXCoreMpLink,'ColourSorterInvalidParametersCombination');

END_ACTION
```

### ConveyorGlobalTypes.typ
```iecst
TYPE
	ConveyorType : 	STRUCT  (*Conveyor Main type*)
		Commands : ConveyorCommadsType;
		Feedbacks : ConveyorFeedbacksType;
		Parameters : ConveyorParametersType;
		Interface : ConveyorInterfaceType;
	END_STRUCT;
	ConveyorCommadsType : 	STRUCT  (*Conveyor Commands type*)
		Enable : BOOL;
		Reset : BOOL;
		Automatic : ConveyorAutomaticCommadsType;
		Manual : ConveyorManualCommadsType;
	END_STRUCT;
	ConveyorFeedbacksType : 	STRUCT  (*Conveyor Feedbacks type*)
		Enabled : BOOL;
		WaitingStart : BOOL;
		Error : BOOL;
		WaitingCap : BOOL;
		InitDone : BOOL;
		AxisHomed : BOOL;
		AxisPowered : BOOL;
		InitPosition : BOOL;
		AxisSpeed : REAL;
		AxisPosition : LREAL;
		NewCapTrigger : BOOL;
		CapsOnConveyor : USINT;
	END_STRUCT;
	ConveyorParametersType : 	STRUCT  (*Conveyor Parameters type*)
		TargetSpeed : REAL := 50;
		Acceleration : REAL := 5000;
	END_STRUCT;
	ConveyorInterfaceType : 	STRUCT  (*Conveyor Interface type*)
		Inputs : ConveyorInterfaceInputsType;
		Outputs : ConveyorInterfaceOutputsType;
	END_STRUCT;
	ConveyorInterfaceOutputsType : 	STRUCT  (*Conveyor Interface Output type*)
		SetSpeed : REAL;
	END_STRUCT;
	ConveyorInterfaceInputsType : 	STRUCT  (*Conveyor Interface Input type*)
		CapInStartPosition : BOOL;
	END_STRUCT;
	ConveyorAutomaticCommadsType : 	STRUCT  (*Conveyor Commands type*)
		Start : BOOL;
		Init : BOOL;
		DecreaseCapCounter : BOOL;
	END_STRUCT;
	ConveyorManualCommadsType : 	STRUCT  (*Conveyor Commands type*)
		Enable : BOOL;
		PowerOn : BOOL;
		Move : BOOL;
		Home : BOOL;
		Speed : REAL := 50;
	END_STRUCT;
END_TYPE
```

### ConveyorGlobalVariables.var
```iecst
VAR
    gConveyor : ConveyorType;
END_VAR
```

### Program Logical/Source/Conveyor/ConveyorProgram (IEC)

#### Main.st - Init, cyclic, exit code
```iecst
//******************************************************************************************************
// Program: 	ConveyorProgram
// Author: 		Andrea Pennisi
// Rev.: 		1.0.0
// Date:		5.12.2023
//
// Description:
// This module is used to deliver the cap from the starting position of the conveyor to the exit.
// An axis is controlled by mappMotion tools. The control is made in velocity.
//******************************************************************************************************
PROGRAM _INIT

    ResetOutputsAction;
    ResetFeedbacksAction;

	Internal.Parameters.Homing.Mode := mcHOMING_ABSOLUTE;

    MachineState.NextState := WAITING_INIT;

END_PROGRAM

PROGRAM _CYCLIC

	MotionAction;

    // Enable module
    IF NOT gConveyor.Commands.Enable THEN
        ResetOutputsAction;
		ResetFeedbacksAction;
		ResetAlarmsAction;
		ResetMotionCommands;
        RETURN;
    END_IF

	IF EDGENEG(gConveyor.Commands.Automatic.Start) THEN
		IF MachineState.NextState <> ERROR THEN
			MachineState.NextState := WAITING_START;
		END_IF
	END_IF

	IF EDGEPOS(gConveyor.Commands.Automatic.Init) THEN
		IF MachineState.NextState <> ERROR THEN
			MachineState.NextState := WAITING_INIT;
		END_IF
	END_IF

	// Alarms
	SetAlarmsAction;

    // Machine state
    MachineStateManagementAction;
    CASE MachineState.ActualState OF

		WAITING_INIT:
			MachineState.TimeoutTimer.PT := T#0S; // Timeout disabled in this state
			IF MachineState.NewTriggerState THEN
				ResetOutputsAction;
				ResetMotionCommands;
			END_IF

			IF gConveyor.Commands.Automatic.Init THEN
				gConveyor.Feedbacks.CapsOnConveyor := 0;
				MachineState.NextState := HOMING;

			ELSIF gConveyor.Commands.Manual.Enable THEN
				MachineState.NextState := MANUALS;

			END_IF

		MANUALS:
			MachineState.TimeoutTimer.PT := T#0S; // Timeout disabled in this state

			Internal.Parameters.Velocity := gConveyor.Commands.Manual.Speed;
			IF Internal.Parameters.Velocity>0 THEN
				Internal.Parameters.Direction := mcDIR_POSITIVE;
			ELSE
				Internal.Parameters.Direction := mcDIR_NEGATIVE;
			END_IF

			Internal.Axis.Home := gConveyor.Commands.Manual.Home AND Internal.Axis.Active AND NOT Internal.Axis.Error;
			IF Internal.Axis.IsHomed THEN
				Internal.Axis.Power := gConveyor.Commands.Manual.PowerOn AND Internal.Axis.Active AND NOT Internal.Axis.Error;
				IF Internal.Axis.PowerOn THEN
					Internal.Axis.MoveVelocity := gConveyor.Commands.Manual.Move AND Internal.Axis.Active AND NOT Internal.Axis.Error;
				ELSE
					Internal.Axis.MoveVelocity := FALSE;
				END_IF
			ELSE
				Internal.Axis.Power := FALSE;
				Internal.Axis.MoveVelocity := FALSE;
			END_IF

			IF NOT gConveyor.Commands.Manual.Enable THEN
				MachineState.NextState := WAITING_INIT;
			END_IF

		HOMING:
			MachineState.TimeoutTimer.PT := T#3S;
			IF Internal.Axis.IsHomed THEN
				Internal.Axis.Home := FALSE;
				MachineState.NextState := POWER_ON;
			ELSE
				Internal.Axis.Home := Internal.Axis.Active AND NOT Internal.Axis.Error;
			END_IF

		POWER_ON:
			MachineState.TimeoutTimer.PT := T#3S;
			Internal.Axis.Power := Internal.Axis.Active AND NOT Internal.Axis.Error;
			IF Internal.Axis.PowerOn THEN
				IF gConveyor.Commands.Automatic.Init THEN
					MachineState.NextState := INIT;
				ELSE
					MachineState.NextState := MOTION;
				END_IF
			END_IF

		INIT:
			MachineState.TimeoutTimer.PT := T#30S;
			IF MachineState.NewTriggerState THEN
				Internal.Parameters.Velocity := gConveyor.Parameters.TargetSpeed;
				Internal.Parameters.Direction := mcDIR_POSITIVE;
			END_IF
			Internal.Axis.MoveAbsolute := Internal.Axis.Active AND NOT Internal.Axis.Error;
			IF Internal.Axis.MoveDone THEN
				Internal.Axis.MoveAbsolute := FALSE;
				MachineState.NextState := WAITING_START;
			END_IF

        WAITING_START:
			MachineState.TimeoutTimer.PT := T#0S; // Timeout disabled in this state
			IF MachineState.NewTriggerState THEN
				ResetMotionCommands;
			END_IF

            IF gConveyor.Commands.Automatic.Start THEN
				MachineState.NextState := POWER_ON;

			ELSIF gConveyor.Commands.Manual.Enable THEN
				MachineState.NextState := MANUALS;
            END_IF

		MOTION:
			MachineState.TimeoutTimer.PT := T#0S; // Timeout disabled in this state
			IF MachineState.NewTriggerState THEN
				Internal.Parameters.Direction := mcDIR_POSITIVE;
			END_IF

			// On-fly velocity change
			IF Internal.Parameters.Velocity <> gConveyor.Parameters.TargetSpeed THEN
				Internal.Parameters.Velocity := gConveyor.Parameters.TargetSpeed;
				Internal.Axis.Update := TRUE;
			ELSIF Internal.Axis.UpdateDone THEN
				Internal.Axis.Update := FALSE;
			END_IF

			Internal.Axis.MoveVelocity := TRUE;

        ERROR:
            MachineState.TimeoutTimer.PT := T#0S; // Timeout disabled in this state
			ResetOutputsAction;
			ResetMotionCommands;
			IF NOT Internal.Error THEN
				MachineState.NextState := WAITING_INIT;
			END_IF

        ELSE
            MachineState.NextState := WAITING_START;

    END_CASE

    FeedbacksUpdateAction;

END_PROGRAM

PROGRAM _EXIT

END_PROGRAM
```

#### Types.typ - Local data types
```iecst
TYPE
	MachineStateType : 	STRUCT  (*Machine state main type*)
		OldState : MachineStateEnum; (*Actual state*)
		ActualState : MachineStateEnum; (*Actual state*)
		NextState : MachineStateEnum; (*Next state*)
		NewTriggerState : BOOL; (*Trigger state change*)
		TimeoutTimer : TON; (*State timeout*)
	END_STRUCT;
	MachineStateEnum :
		( (*Machine State enumeration*)
		WAITING_INIT, (*WAITING state*)
		MANUALS,
		WAITING_START,
		HOMING,
		POWER_ON,
		INIT,
		MOTION,
		ERROR (*ERROR state*)
		);
	InternalType : 	STRUCT
		Axis : MpAxisBasic;
		Parameters : MpAxisBasicParType;
		Error : BOOL;
	END_STRUCT;
END_TYPE
```

#### Variables.var - Local variables
```iecst
VAR
	MachineState : MachineStateType;
	Internal : InternalType;
END_VAR
```

#### Actions.st
```iecst
ACTION FeedbacksUpdateAction:

    gConveyor.Feedbacks.Enabled := TRUE;
    gConveyor.Feedbacks.WaitingStart := MachineState.ActualState = WAITING_START;
    gConveyor.Feedbacks.Error := MachineState.ActualState = ERROR;
	gConveyor.Feedbacks.WaitingCap := MachineState.ActualState = MOTION AND (gConveyor.Feedbacks.CapsOnConveyor = 0);
	gConveyor.Feedbacks.AxisHomed := Internal.Axis.IsHomed;
	gConveyor.Feedbacks.AxisPowered := Internal.Axis.PowerOn;
	gConveyor.Feedbacks.InitPosition := ABS(Internal.Axis.Position - Internal.Parameters.Position)<0.1;
	gConveyor.Feedbacks.InitDone := gConveyor.Feedbacks.InitPosition AND gConveyor.Commands.Automatic.Init;
	gConveyor.Feedbacks.AxisSpeed := Internal.Axis.Velocity;
	gConveyor.Feedbacks.AxisPosition := Internal.Axis.Position;

	IF EDGEPOS(gConveyor.Interface.Inputs.CapInStartPosition) AND gConveyor.Commands.Automatic.Start THEN
		gConveyor.Feedbacks.CapsOnConveyor := gConveyor.Feedbacks.CapsOnConveyor + 1;

	ELSIF gConveyor.Interface.Inputs.CapInStartPosition AND gConveyor.Commands.Automatic.Start AND gConveyor.Feedbacks.CapsOnConveyor = 0 THEN
		gConveyor.Feedbacks.CapsOnConveyor := gConveyor.Feedbacks.CapsOnConveyor + 1;

	END_IF

	IF EDGEPOS(gConveyor.Commands.Automatic.DecreaseCapCounter) THEN
		IF gConveyor.Feedbacks.CapsOnConveyor > 1 THEN
			gConveyor.Feedbacks.CapsOnConveyor := gConveyor.Feedbacks.CapsOnConveyor - 1;
		ELSE
			gConveyor.Feedbacks.CapsOnConveyor := 0;
		END_IF
	END_IF

END_ACTION

ACTION ResetOutputsAction:

	memset(ADR(gConveyor.Interface.Outputs),0,SIZEOF(gConveyor.Interface.Outputs));

END_ACTION

ACTION ResetMotionCommands:
	Internal.Axis.Power := FALSE;
	Internal.Axis.Home := FALSE;
	Internal.Axis.MoveVelocity := FALSE;
	Internal.Axis.MoveAbsolute := FALSE;
	Internal.Axis.Update := FALSE;
END_ACTION

ACTION ResetFeedbacksAction:

    memset(ADR(gConveyor.Feedbacks),0,SIZEOF(gConveyor.Feedbacks));

END_ACTION

ACTION MachineStateManagementAction:

    // Machine state timeout check
    MachineState.TimeoutTimer(IN := MachineState.TimeoutTimer.PT <> T#0S AND NOT MachineState.NewTriggerState);

    // Machine state change state logic
    MachineState.NewTriggerState := (MachineState.ActualState <> MachineState.NextState);
    IF MachineState.NewTriggerState THEN
        MachineState.OldState := MachineState.ActualState;
    END_IF
    MachineState.ActualState := MachineState.NextState;

END_ACTION

ACTION SetAlarmsAction:

	IF gConveyor.Commands.Reset THEN
		Internal.Error := FALSE;
	END_IF

	IF MachineState.TimeoutTimer.Q THEN

		CASE MachineState.ActualState OF
			HOMING: MpAlarmXSet(gAlarmXCoreMpLink,'ConveyorTimeoutHoming'); // Edge alarm!
			POWER_ON: MpAlarmXSet(gAlarmXCoreMpLink,'ConveyorTimeoutPowerOn'); // Edge alarm!
			INIT: MpAlarmXSet(gAlarmXCoreMpLink,'ConveyorInitFail'); // Edge alarm!
		END_CASE

		Internal.Error := TRUE;
		MachineState.NextState := ERROR;
	END_IF

	// ConveyorAxisError
	IF Internal.Axis.Error THEN
		MpAlarmXSet(gAlarmXCoreMpLink,'ConveyorAxisError');
		Internal.Error := TRUE;
		MachineState.NextState := ERROR;
	ELSE
		MpAlarmXReset(gAlarmXCoreMpLink,'ConveyorAxisError');
	END_IF

	// ConveyorTooManyCaps
	IF gConveyor.Commands.Reset THEN
		gConveyor.Feedbacks.CapsOnConveyor := 0;
	END_IF
	IF gConveyor.Feedbacks.CapsOnConveyor > 1 THEN
		MpAlarmXSet(gAlarmXCoreMpLink,'ConveyorTooManyCaps');
		Internal.Error := TRUE;
		MachineState.NextState := ERROR;
	ELSE
		MpAlarmXReset(gAlarmXCoreMpLink,'ConveyorTooManyCaps');
	END_IF
END_ACTION

ACTION ResetAlarmsAction:

	MpAlarmXReset(gAlarmXCoreMpLink,'ConveyorAxisError');

END_ACTION
```

#### MotionAction.ld
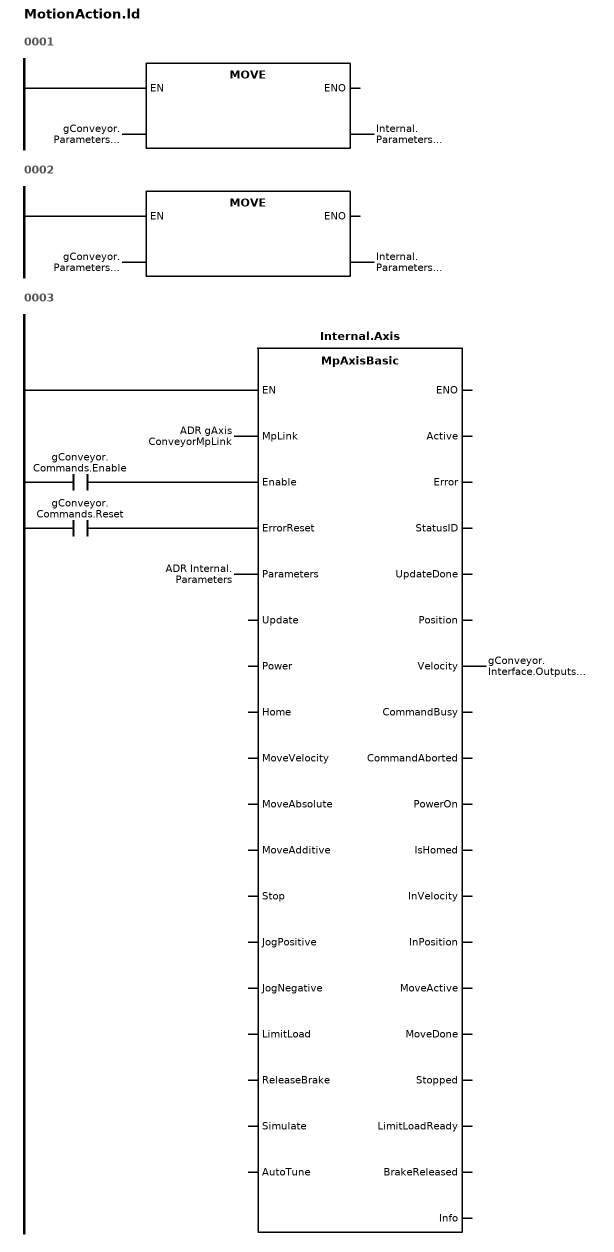
Ladder, written as Structured Text:
```iecst
ACTION MotionAction:
(* Network 1 *)
Internal.Parameters.Deceleration := gConveyor.Parameters.Acceleration;

(* Network 2 *)
Internal.Parameters.Acceleration := gConveyor.Parameters.Acceleration;

(* Network 3 *)
Internal.Axis(MpLink := ADR(gAxisConveyorMpLink), Enable := gConveyor.Commands.Enable, ErrorReset := gConveyor.Commands.Reset, Parameters := ADR(Internal.Parameters));
gConveyor.Interface.Outputs.SetSpeed := Internal.Axis.Velocity;
END_ACTION
```

### PuncherGlobalTypes.typ
```iecst
TYPE
	PuncherType : 	STRUCT  (*Puncher Main type*)
		Commands : PuncherCommadsType;
		Feedbacks : PuncherFeedbacksType;
		Parameters : PuncherParametersType;
		Interface : PuncherInterfaceType;
	END_STRUCT;
	PuncherCommadsType : 	STRUCT  (*Puncher Commands type*)
		Enable : BOOL;
		Reset : BOOL;
		Automatic : PuncherAutomaticCommadsType;
		Manual : PuncherManualCommadsType;
	END_STRUCT;
	PuncherFeedbacksType : 	STRUCT  (*Puncher Feedbacks type*)
		Enabled : BOOL;
		WaitingStart : BOOL;
		Error : BOOL;
		OnSyncMotion : BOOL;
		WaitingCap : BOOL;
		PunchCapDone : BOOL;
		InitDone : BOOL;
		InitPosition : BOOL;
		AxisSpeed : REAL;
		AxisPosition : LREAL;
		AxisHomed : BOOL;
		AxisPowered : BOOL;
	END_STRUCT;
	PuncherParametersType : 	STRUCT  (*Puncher Parameters type*)
		Offset : REAL := 25;
		Speed : REAL := 10000;
		Acceleration : REAL := 20000;
	END_STRUCT;
	PuncherInterfaceType : 	STRUCT  (*Puncher Interface type*)
		Inputs : PuncherInterfaceInputsType;
		Outputs : PuncherInterfaceOutputsType;
	END_STRUCT;
	PuncherInterfaceOutputsType : 	STRUCT  (*Puncher Interface Output type*)
		PunchForward : BOOL;
		SetPosition : LREAL;
	END_STRUCT;
	PuncherInterfaceInputsType : 	STRUCT  (*Puncher Interface Input type*)
		ActualPosition : REAL;
		PunchIsForward : BOOL;
		PunchIsBackward : BOOL;
	END_STRUCT;
	PuncherAutomaticCommadsType : 	STRUCT  (*Puncher Commands type*)
		Start : BOOL;
		Init : BOOL;
		PunchCap : BOOL;
	END_STRUCT;
	PuncherManualCommadsType : 	STRUCT  (*Puncher Commands type*)
		Enable : BOOL;
		PuncherForward : BOOL;
		Position : LREAL;
		Speed : REAL := 50;
		PowerOn : BOOL;
		Move : BOOL;
		Home : BOOL;
	END_STRUCT;
END_TYPE
```

### PuncherGlobalVariables.var
```iecst
VAR
	gPuncher : PuncherType;
END_VAR
```

### Program Logical/Source/Puncher/PuncherProgram (IEC)

#### Main.st - Init, cyclic, exit code
```iecst
//******************************************************************************************************
// Program: 	PuncherProgram
// Author: 		Andrea Pennisi
// Rev.: 		1.0.0
// Date:		5.12.2023
//
// Description:
// This module is used to punch the the cap.
// An axis is controlled by mappMotion tools. The control is made by a cam linked to the Conveyor module axis.
//******************************************************************************************************
PROGRAM _INIT

    ResetOutputsAction;
    ResetFeedbacksAction;

	Internal.Parameters.Homing.Mode := mcHOMING_DIRECT;

	Internal.Offset.AdvancedParameters.ShiftMode := mcSHIFT_ABSOLUTE;
	Internal.Offset.Enable := TRUE;

    MachineState.NextState := WAITING_INIT;

END_PROGRAM

PROGRAM _CYCLIC

	MotionAction;

    // Enable module
    IF NOT gPuncher.Commands.Enable THEN
        ResetOutputsAction;
		ResetFeedbacksAction;
		ResetAlarmsAction;
		ResetMotionCommands;
        RETURN;
    END_IF

	IF EDGENEG(gPuncher.Commands.Automatic.Start) THEN
		IF MachineState.NextState <> ERROR THEN
			MachineState.NextState := WAITING_START;
		END_IF
	END_IF

	IF EDGEPOS(gPuncher.Commands.Automatic.Init) THEN
		IF MachineState.NextState <> ERROR THEN
			MachineState.NextState := WAITING_INIT;
		END_IF
	END_IF

	// Alarms
	SetAlarmsAction;

    // Machine state
    MachineStateManagementAction;
    CASE MachineState.ActualState OF

		WAITING_INIT:
			MachineState.TimeoutTimer.PT := T#0S; // Timeout disabled in this state
			IF MachineState.NewTriggerState THEN
				ResetOutputsAction;
				ResetMotionCommands;
				Internal.CamStartTrigger := FALSE;
			END_IF

			IF gPuncher.Commands.Automatic.Init THEN
				MachineState.NextState := HOMING;

			ELSIF gPuncher.Commands.Manual.Enable THEN
				MachineState.NextState := MANUAL;

			END_IF

		MANUAL:
			MachineState.TimeoutTimer.PT := T#0S; // Timeout disabled in this state

			Internal.Parameters.Velocity := gPuncher.Commands.Manual.Speed;
			Internal.Parameters.Position := gPuncher.Commands.Manual.Position;

			gPuncher.Interface.Outputs.PunchForward := gPuncher.Commands.Manual.PuncherForward;

			Internal.Axis.Home := gPuncher.Commands.Manual.Home AND Internal.Axis.Active AND NOT Internal.Axis.Error;
			IF Internal.Axis.IsHomed THEN
				Internal.Axis.Power := gPuncher.Commands.Manual.PowerOn AND Internal.Axis.Active AND NOT Internal.Axis.Error;
				IF Internal.Axis.PowerOn THEN
					Internal.Axis.MoveAbsolute := gPuncher.Commands.Manual.Move AND Internal.Axis.Active AND NOT Internal.Axis.Error;
				ELSE
					Internal.Axis.MoveAbsolute := FALSE;
				END_IF
			ELSE
				Internal.Axis.Power := FALSE;
				Internal.Axis.MoveAbsolute := FALSE;
			END_IF

			IF NOT gPuncher.Commands.Manual.Enable THEN
				MachineState.NextState := WAITING_INIT;
			END_IF

		HOMING:
			MachineState.TimeoutTimer.PT := T#3S;
			IF Internal.Axis.IsHomed THEN
				Internal.Axis.Home := FALSE;
				MachineState.NextState := POWER_ON;
			ELSE
				Internal.Axis.Home := Internal.Axis.Active AND NOT Internal.Axis.Error;
			END_IF

		POWER_ON:
			MachineState.TimeoutTimer.PT := T#3S;

			Internal.Axis.Power := Internal.Axis.Active AND NOT Internal.Axis.Error;
			IF Internal.Axis.PowerOn THEN
				IF gPuncher.Commands.Automatic.Init THEN
					MachineState.NextState := INIT;
				ELSE
					MachineState.NextState := ACTIVATE_CAM;
				END_IF
			END_IF

		INIT:
			MachineState.TimeoutTimer.PT := T#15S;
			Internal.Parameters.Position := 0;
			Internal.Parameters.Velocity := gPuncher.Parameters.Speed;
			Internal.Axis.MoveAbsolute := Internal.Axis.Active AND NOT Internal.Axis.Error;
			IF Internal.Axis.MoveDone THEN
				Internal.OffsetToDo := TRUE;
				Internal.Axis.MoveAbsolute := FALSE;
				MachineState.NextState := WAITING_START;
			END_IF

        WAITING_START:
			MachineState.TimeoutTimer.PT := T#0S; // Timeout disabled in this state
			IF MachineState.NewTriggerState THEN
				ResetMotionCommands;
				Internal.Parameters.Velocity := gPuncher.Parameters.Speed;
			END_IF

			IF gPuncher.Commands.Automatic.Start THEN
				gPuncher.Feedbacks.PunchCapDone := FALSE;
				MachineState.NextState := POWER_ON;

			ELSIF gPuncher.Commands.Manual.Enable THEN
				MachineState.NextState := MANUAL;
            END_IF

		ACTIVATE_CAM:
			MachineState.TimeoutTimer.PT := T#0S; // Timeout disabled in this state
			Internal.Cam.Enable := TRUE;
			Internal.Cam.Start := TRUE;
			IF Internal.Axis.Info.PLCopenState = mcAXIS_SYNCHRONIZED_MOTION THEN
				MachineState.NextState := WAITING_CAP;
			END_IF

		WAITING_CAP:
			MachineState.TimeoutTimer.PT := T#0S; // Timeout disabled in this state
			IF gPuncher.Commands.Automatic.PunchCap THEN
				gPuncher.Feedbacks.PunchCapDone := FALSE;
				Internal.CamStartTrigger := TRUE;
			END_IF

			IF Internal.Cam.InCam AND Internal.Cam.ActualStateIndex = 1 THEN // Syncronized motion
				Internal.CamStartTrigger := FALSE;
				MachineState.NextState := PUNCH_FORWARD;
			END_IF

		PUNCH_FORWARD:
			MachineState.TimeoutTimer.PT := T#3S;

			gPuncher.Interface.Outputs.PunchForward := TRUE;
			IF gPuncher.Interface.Inputs.PunchIsForward THEN
				MachineState.NextState := PUNCHING;
			END_IF

		PUNCHING:
			MachineState.TimeoutTimer.PT := T#15S;

			IF Internal.Cam.ActualStateIndex <> 1 THEN
				gPuncher.Interface.Outputs.PunchForward := FALSE;
				MachineState.NextState := PUNCH_BACKWARD;
			END_IF

		PUNCH_BACKWARD:
			MachineState.TimeoutTimer.PT := T#3S;

			IF gPuncher.Interface.Inputs.PunchIsBackward THEN
				gPuncher.Feedbacks.PunchCapDone := TRUE;
				MachineState.NextState := WAITING_CAP;
			END_IF

        ERROR:
            MachineState.TimeoutTimer.PT := T#0S; // Timeout disabled in this state
			ResetOutputsAction;
			ResetMotionCommands;
			IF NOT Internal.Error THEN
				MachineState.NextState := WAITING_INIT;
			END_IF

        ELSE
            MachineState.NextState := WAITING_START;

    END_CASE

	OffsetManagement;

    FeedbacksUpdateAction;

END_PROGRAM

PROGRAM _EXIT

END_PROGRAM
```

#### Types.typ - Local data types
```iecst
TYPE
	MachineStateType : 	STRUCT  (*Machine state main type*)
		OldState : MachineStateEnum; (*Actual state*)
		ActualState : MachineStateEnum; (*Actual state*)
		NextState : MachineStateEnum; (*Next state*)
		NewTriggerState : BOOL; (*Trigger state change*)
		TimeoutTimer : TON; (*State timeout*)
	END_STRUCT;
	MachineStateEnum :
		( (*Machine State enumeration*)
		WAITING_INIT,
		MANUAL,
		WAITING_START, (*WAITING state*)
		HOMING,
		POWER_ON, (*INIT state*)
		INIT,
		ACTIVATE_CAM,
		WAITING_CAP,
		PUNCH_FORWARD,
		PUNCHING,
		PUNCH_BACKWARD,
		ERROR (*ERROR state*)
		);
	InternalType : 	STRUCT
		Axis : MpAxisBasic;
		Parameters : MpAxisBasicParType;
		Cam : MC_BR_CamAutomatCommand;
		Offset : MC_BR_Offset;
		LastOffset : LREAL;
		CamStartTrigger : BOOL;
		Error : BOOL;
		OffsetToDo : BOOL;
	END_STRUCT;
END_TYPE
```

#### Variables.var - Local variables
```iecst
VAR
	MachineState : MachineStateType;
	Internal : InternalType;
END_VAR
```

#### Actions.st
```iecst
ACTION FeedbacksUpdateAction:

    gPuncher.Feedbacks.Enabled := TRUE;
    gPuncher.Feedbacks.WaitingStart := (MachineState.ActualState = WAITING_START);
	gPuncher.Feedbacks.Error := (MachineState.ActualState = ERROR);
	gPuncher.Feedbacks.OnSyncMotion := Internal.Cam.InCam;
	gPuncher.Feedbacks.WaitingCap := (Internal.Cam.ActualStateIndex = 0) AND (MachineState.ActualState = WAITING_CAP);
	gPuncher.Feedbacks.InitPosition := ABS(Internal.Axis.Position - Internal.Parameters.Position)<0.1;
	gPuncher.Feedbacks.InitDone := gPuncher.Feedbacks.InitPosition AND gPuncher.Commands.Automatic.Init;
	gPuncher.Feedbacks.AxisHomed := Internal.Axis.IsHomed;
	gPuncher.Feedbacks.AxisPowered := Internal.Axis.PowerOn;
	gPuncher.Feedbacks.AxisSpeed := Internal.Axis.Velocity;
	gPuncher.Feedbacks.AxisPosition := Internal.Axis.Position;

END_ACTION

ACTION ResetOutputsAction:

    memset(ADR(gPuncher.Interface.Outputs),0,SIZEOF(gPuncher.Interface.Outputs));

END_ACTION

ACTION ResetFeedbacksAction:

    memset(ADR(gPuncher.Feedbacks),0,SIZEOF(gPuncher.Feedbacks));

END_ACTION

ACTION ResetMotionCommands:
	Internal.Axis.Power := FALSE;
	Internal.Axis.Home := FALSE;
	Internal.Axis.MoveVelocity := FALSE;
	Internal.Axis.MoveAbsolute := FALSE;

	Internal.Cam.Enable := FALSE;
	Internal.Cam.Start := FALSE;

	Internal.Offset.Enable := FALSE;
	Internal.Offset.StartShift := FALSE;
END_ACTION

ACTION MachineStateManagementAction:

    // Machine state timeout check
    MachineState.TimeoutTimer(IN := MachineState.TimeoutTimer.PT <> T#0S AND NOT MachineState.NewTriggerState);

    // Machine state change state logic
    MachineState.NewTriggerState := (MachineState.ActualState <> MachineState.NextState);
    IF MachineState.NewTriggerState THEN
        MachineState.OldState := MachineState.ActualState;
    END_IF
    MachineState.ActualState := MachineState.NextState;

END_ACTION

ACTION SetAlarmsAction:

	IF gPuncher.Commands.Reset THEN
		Internal.Error := FALSE;
	END_IF

	IF MachineState.TimeoutTimer.Q THEN

		CASE MachineState.ActualState OF
			HOMING: MpAlarmXSet(gAlarmXCoreMpLink,'PuncherTimeoutHoming'); // Edge alarm!
			POWER_ON: MpAlarmXSet(gAlarmXCoreMpLink,'PuncherTimeoutPowerOn'); // Edge alarm!
			PUNCH_FORWARD: MpAlarmXSet(gAlarmXCoreMpLink,'PuncherTimeoutPunchForward'); // Edge alarm!
			PUNCH_BACKWARD: MpAlarmXSet(gAlarmXCoreMpLink,'PuncherTimeoutPunchBackward'); // Edge alarm!
			ACTIVATE_CAM: MpAlarmXSet(gAlarmXCoreMpLink,'PuncherAxisTimeout'); // Edge alarm!
			PUNCHING: MpAlarmXSet(gAlarmXCoreMpLink,'PuncherAxisTimeout'); // Edge alarm!
		END_CASE

		Internal.Error := TRUE;
		MachineState.NextState := ERROR;
	END_IF

	IF Internal.Axis.Error OR Internal.Cam.Error OR Internal.Offset.Error THEN
		MpAlarmXSet(gAlarmXCoreMpLink,'PuncherAxisError');
		Internal.Error := TRUE;
		MachineState.NextState := ERROR;
	ELSE
		MpAlarmXReset(gAlarmXCoreMpLink,'PuncherAxisError');
	END_IF

	IF gPuncher.Interface.Inputs.PunchIsForward AND gPuncher.Interface.Inputs.PunchIsBackward THEN
		MpAlarmXSet(gAlarmXCoreMpLink,'PuncherInvalidSensorsCombination');
		Internal.Error := TRUE;
		MachineState.NextState := ERROR;
	ELSE
		MpAlarmXReset(gAlarmXCoreMpLink,'PuncherInvalidSensorsCombination');
	END_IF

END_ACTION

ACTION ResetAlarmsAction:

	MpAlarmXReset(gAlarmXCoreMpLink,'PuncherInvalidSensorsCombination');

END_ACTION

ACTION OffsetManagement:

	Internal.Offset.Enable := Internal.Axis.Info.PLCopenState = mcAXIS_SYNCHRONIZED_MOTION;
	Internal.Offset.StartShift := (Internal.OffsetToDo OR Internal.LastOffset <> gPuncher.Parameters.Offset) AND Internal.Offset.Valid;
	Internal.LastOffset := gPuncher.Parameters.Offset;
	IF Internal.OffsetToDo AND Internal.Offset.StartShift THEN
		Internal.OffsetToDo := FALSE;
	END_IF

END_ACTION
```

#### MotionAction.ld
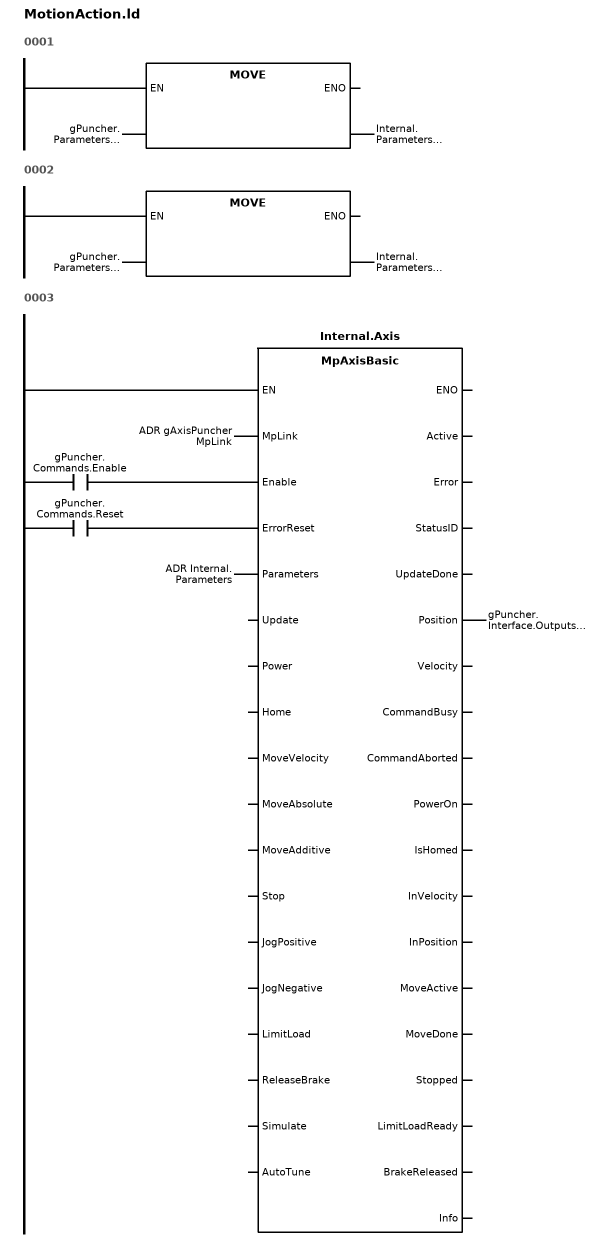
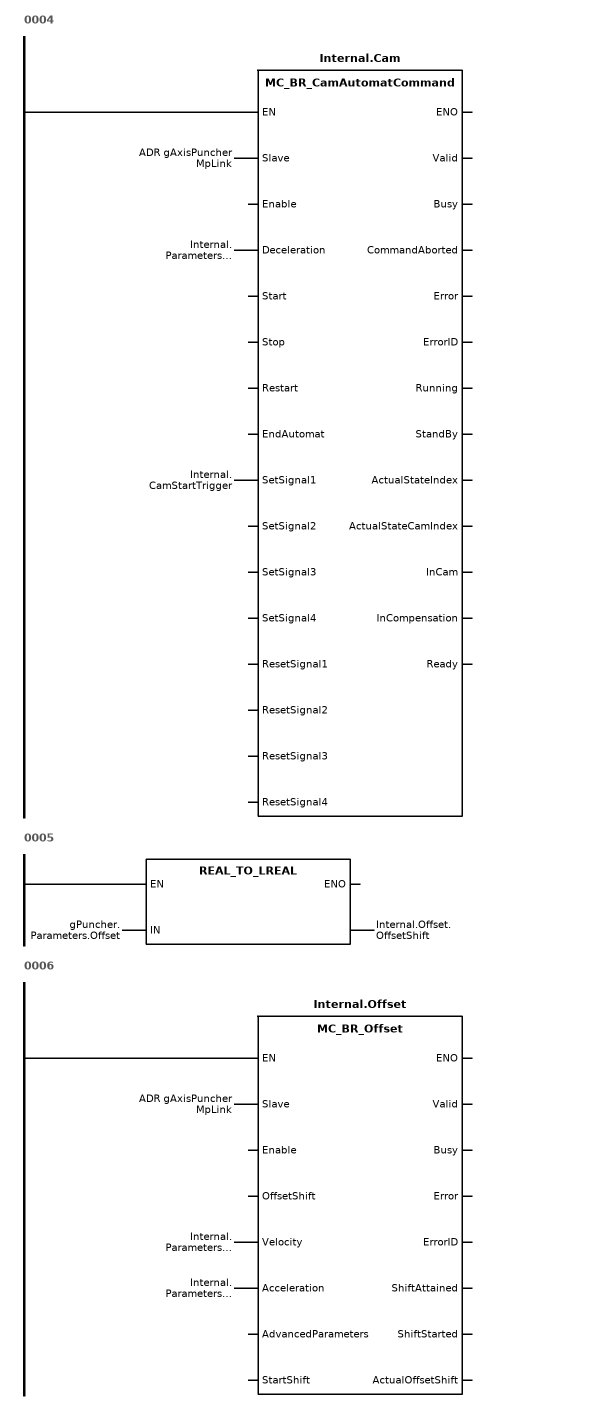
Ladder, written as Structured Text:
```iecst
ACTION MotionAction:
(* Network 1 *)
Internal.Parameters.Deceleration := gPuncher.Parameters.Acceleration;

(* Network 2 *)
Internal.Parameters.Acceleration := gPuncher.Parameters.Acceleration;

(* Network 3 *)
Internal.Axis(MpLink := ADR(gAxisPuncherMpLink), Enable := gPuncher.Commands.Enable, ErrorReset := gPuncher.Commands.Reset, Parameters := ADR(Internal.Parameters));
gPuncher.Interface.Outputs.SetPosition := Internal.Axis.Position;

(* Network 4 *)
Internal.Cam(Slave := ADR(gAxisPuncherMpLink), Deceleration := Internal.Parameters.Deceleration, SetSignal1 := Internal.CamStartTrigger);

(* Network 5 *)
Internal.Offset.OffsetShift := REAL_TO_LREAL(gPuncher.Parameters.Offset);

(* Network 6 *)
Internal.Offset(Slave := ADR(gAxisPuncherMpLink), Velocity := Internal.Parameters.Velocity, Acceleration := Internal.Parameters.Acceleration);
END_ACTION
```

### MainMachineGlobalTypes.typ
```iecst
TYPE
	MainMachineType : 	STRUCT  (*MainMachine Main type*)
		Commands : MainMachineCommadsType;
		Feedbacks : MainMachineFeedbacksType;
		Parameters : MainMachineParametersType;
		Statistics : MainMachineStatisticsType;
	END_STRUCT;
	MainMachineCommadsType : 	STRUCT  (*MainMachine Commands type*)
		LinkMode : BOOL;
		Reset : BOOL;
		ClearStats : BOOL;
		Automatic : MainMachineAutomaticCommadsType;
		Manual : MainMachineManualCommadsType;
	END_STRUCT;
	MainMachineFeedbacksType : 	STRUCT  (*MainMachine Feedbacks type*)
		WaitingStart : BOOL;
		Started : BOOL;
		Stopping : BOOL;
		Error : BOOL;
		AutomaticMode : BOOL;
		LinkOk : BOOL;
		ManualMode : BOOL;
		InitDone : BOOL;
		WaitModeSelection : BOOL;
		WaitingInit : BOOL;
		NewCapOnWork : BOOL;
		ClearStatsDone : BOOL;
		Initializing : BOOL;
		WaitingModulesReady : BOOL;
		PunchingCap : BOOL;
		SortingCap : BOOL;
		DeliveringCap : BOOL;
		WaitingCap : BOOL;
		AskRemoveCaps : BOOL;
		CapsOnConveyor : USINT;
	END_STRUCT;
	MainMachineParametersType : 	STRUCT  (*MainMachine Parameters type*)
		PuncherEnable : BOOL := TRUE;
	END_STRUCT;
	MainMachineStatisticsType : 	STRUCT
		CapsCounter : UDINT;
		CurrentCapWorkingTime : TIME;
		LastCapWorkingTime : TIME;
		AverageCapWorkingTime : TIME;
	END_STRUCT;
	MainMachineAutomaticCommadsType : 	STRUCT  (*MainMachine Commands type*)
		Enable : BOOL;
		Init : BOOL;
		Start : BOOL;
		CapsRemoved : BOOL;
	END_STRUCT;
	MainMachineManualCommadsType : 	STRUCT  (*MainMachine Commands type*)
		Enable : BOOL;
	END_STRUCT;
END_TYPE
```

### MainMachineGlobalVariables.var
```iecst
VAR
	gMainMachine : MainMachineType;
END_VAR
VAR CONSTANT
	STATS_HISTORY_MAX_INDEX : USINT := 9;
END_VAR
```

### Program Logical/Source/MainMachine/MainMachineProgram (IEC)

#### Main.st - Init, cyclic, exit code
```iecst
PROGRAM _INIT

	EnableModules;

    MachineState.NextState := WAITING_MODE_SELECTION;

END_PROGRAM

PROGRAM _CYCLIC

	// Master communication management
	PickingStationCommunication;

	// Alarms
	SetAlarmsAction;

	// Check stop reaction
	IF MpAlarmXCheckReaction(gAlarmXCoreMpLink,'STOP')
		OR (MpAlarmXCheckReaction(gAlarmXCoreMpLink,'STOP_ON_PHASE') AND NOT gMainMachine.Feedbacks.Started) THEN
		MachineState.NextState := ERROR;
	END_IF

	// Machine state
	MachineStateManagementAction;
	CASE MachineState.ActualState OF

		WAITING_MODE_SELECTION:
			MachineState.TimeoutTimer.PT := T#0S; // Timeout disabled in this state
			IF MachineState.NewTriggerState THEN
				StopModules;
			END_IF

			IF gMainMachine.Commands.Automatic.Enable THEN
				MachineState.NextState := AUTO_WAITING_INIT;

			ELSIF gMainMachine.Commands.Manual.Enable THEN
				MachineState.NextState := MANUAL;
			END_IF

		MANUAL:
			MachineState.TimeoutTimer.PT := T#0S; // Timeout disabled in this state
			IF MachineState.NewTriggerState THEN
				ResetModulesManualCommands;
			END_IF

			gColourSorter.Commands.Manual.Enable := TRUE;
			gConveyor.Commands.Manual.Enable := TRUE;
			gPuncher.Commands.Manual.Enable := TRUE;

			IF NOT gMainMachine.Commands.Manual.Enable THEN
				MachineState.NextState := WAITING_MODE_SELECTION;
			END_IF

		AUTO_WAITING_INIT:
			MachineState.TimeoutTimer.PT := T#0S; // Timeout disabled in this state
			IF MachineState.NewTriggerState THEN
				gMainMachine.Feedbacks.InitDone := FALSE;
			END_IF

			IF NOT gMainMachine.Commands.Automatic.Enable THEN
				MachineState.NextState := WAITING_MODE_SELECTION;

			ELSIF gMainMachine.Commands.Automatic.Init THEN
				MachineState.NextState := AUTO_INITIALIZING;

			END_IF

		AUTO_INITIALIZING:
			MachineState.TimeoutTimer.PT := T#30S;
			IF MachineState.NewTriggerState THEN
				InitModules;
			END_IF

			IF gColourSorter.Feedbacks.InitDone
				AND gConveyor.Feedbacks.InitDone
				AND gPuncher.Feedbacks.InitDone
				AND (gPickingStation.Outputs.InitDone OR NOT gMainMachine.Commands.LinkMode) THEN

				gMainMachine.Feedbacks.InitDone := TRUE;
				MachineState.NextState := AUTO_WAITING_START;

			END_IF

		AUTO_WAITING_START:
			MachineState.TimeoutTimer.PT := T#0S; // Timeout disabled in this state
			IF MachineState.NewTriggerState THEN
				StopModules;
			END_IF

			IF NOT gMainMachine.Commands.Automatic.Enable THEN
				MachineState.NextState := WAITING_MODE_SELECTION;

			ELSIF gMainMachine.Commands.LinkMode AND NOT gPickingStation.Outputs.WaitingStart THEN // Picking station was linked after this station initialization
				MachineState.NextState := WAITING_MODE_SELECTION;

			ELSIF gMainMachine.Commands.Automatic.Start THEN
				StartModules;
				MachineState.NextState := AUTO_WAITING_MODULES_READY;

			END_IF

		AUTO_WAITING_MODULES_READY:
			MachineState.TimeoutTimer.PT := T#0S; // Timeout disabled in this state
			IF MachineState.NewTriggerState THEN
				Internal.LastCapCounter := gConveyor.Feedbacks.CapsOnConveyor;
				gConveyor.Commands.Automatic.DecreaseCapCounter := TRUE;
				gMainMachine.Feedbacks.NewCapOnWork := FALSE;
			END_IF

			IF NOT gMainMachine.Commands.Automatic.Start AND (NOT gPickingStation.Outputs.Started OR NOT gMainMachine.Commands.LinkMode) THEN

				gConveyor.Commands.Automatic.DecreaseCapCounter := FALSE;
				MachineState.NextState := WAITING_MODE_SELECTION;

			ELSIF Internal.LastCapCounter <> gConveyor.Feedbacks.CapsOnConveyor OR gConveyor.Feedbacks.CapsOnConveyor = 0 THEN

				IF gColourSorter.Feedbacks.WaitingCap
					AND gConveyor.Feedbacks.WaitingCap
					AND (gPuncher.Feedbacks.WaitingCap OR NOT gPuncher.Commands.Automatic.Start)
					AND (gPickingStation.Outputs.Started OR NOT gMainMachine.Commands.LinkMode) THEN

					gConveyor.Commands.Automatic.DecreaseCapCounter := FALSE;
					MachineState.NextState := AUTO_WAITING_CAP;
				END_IF
			END_IF

		AUTO_WAITING_CAP:
			MachineState.TimeoutTimer.PT := T#0S; // Timeout disabled in this state

			IF MpAlarmXCheckReaction(gAlarmXCoreMpLink,'STOP_ON_PHASE') THEN
				MachineState.NextState := ERROR;

			ELSIF NOT gMainMachine.Commands.Automatic.Start AND (NOT gPickingStation.Outputs.Started OR NOT gMainMachine.Commands.LinkMode) THEN

				MachineState.NextState := WAITING_MODE_SELECTION;

			ELSIF gConveyor.Feedbacks.CapsOnConveyor = 1 THEN
				gMainMachine.Feedbacks.NewCapOnWork := TRUE;
				gPuncher.Commands.Automatic.PunchCap := TRUE;
				MachineState.NextState := AUTO_DELIVERING_AND_PUNCHING_CAP;
			END_IF

		AUTO_DELIVERING_AND_PUNCHING_CAP:
			MachineState.TimeoutTimer.PT := T#15S;
			IF NOT gPuncher.Feedbacks.WaitingCap THEN
				gPuncher.Commands.Automatic.PunchCap := FALSE;
			END_IF

			IF gPuncher.Commands.Automatic.Start THEN

				IF NOT gPuncher.Commands.Automatic.PunchCap AND gPuncher.Feedbacks.PunchCapDone THEN
					MachineState.NextState := AUTO_SORTING_CAP;
				END_IF

			ELSE
				MachineState.NextState := AUTO_SORTING_CAP;
			END_IF

		AUTO_SORTING_CAP:
			MachineState.TimeoutTimer.PT := T#15S;

			IF EDGEPOS(gColourSorter.Feedbacks.CapSorted) THEN
				MachineState.NextState := AUTO_WAITING_MODULES_READY;
			END_IF

		AUTO_WAITING_PICKUP_STATION_STOP:
			MachineState.TimeoutTimer.PT := T#0S; // Timeout disabled in this state
			gPickingStation.Inputs.Start := FALSE;
			IF NOT gPickingStation.Outputs.Started OR NOT gMainMachine.Commands.LinkMode THEN
				MachineState.NextState := AUTO_WAITING_START;
			END_IF

		ERROR:
			MachineState.TimeoutTimer.PT := T#0S; // Timeout disabled in this state
			IF MachineState.NewTriggerState THEN
				StopModules;
				ResetModulesManualCommands;
				gMainMachine.Commands.Reset := FALSE;
			END_IF

			IF EDGE(gMainMachine.Commands.Automatic.Init) THEN
				gMainMachine.Commands.Reset := gMainMachine.Commands.Automatic.Init; // User can reset alarms with init command
			END_IF

			gColourSorter.Commands.Reset := gMainMachine.Commands.Reset;
			gConveyor.Commands.Reset := gMainMachine.Commands.Reset;
			gPuncher.Commands.Reset := gMainMachine.Commands.Reset;
			gPickingStation.Inputs.Reset := gMainMachine.Commands.Reset;

			IF gMainMachine.Commands.Reset THEN
				gAlarms.MpAlarmXListUIConnect.AcknowledgeAll := TRUE;
			END_IF

			IF NOT MpAlarmXCheckReaction(gAlarmXCoreMpLink,'STOP')
				AND NOT MpAlarmXCheckReaction(gAlarmXCoreMpLink,'STOP_ON_PHASE')
				AND (NOT gPickingStation.Outputs.Error OR NOT gMainMachine.Commands.LinkMode) THEN

				gMainMachine.Commands.Reset := FALSE;
				MachineState.NextState := WAITING_MODE_SELECTION;
			END_IF

		ELSE
			MachineState.NextState := WAITING_MODE_SELECTION;

	END_CASE

	PickingStationAction;

	FeedbacksUpdateAction;

	StatisticsAction;

END_PROGRAM

PROGRAM _EXIT

END_PROGRAM
```

#### Types.typ - Local data types
```iecst
TYPE
	MachineStateType : 	STRUCT  (*Machine state main type*)
		OldState : MachineStateEnum; (*Actual state*)
		ActualState : MachineStateEnum; (*Actual state*)
		NextState : MachineStateEnum; (*Next state*)
		NewTriggerState : BOOL; (*Trigger state change*)
		TimeoutTimer : TON; (*State timeout*)
	END_STRUCT;
	MachineStateEnum :
		( (*Machine State enumeration*)
		WAITING_MODE_SELECTION,
		MANUAL,
		AUTO_WAITING_INIT,
		AUTO_INITIALIZING,
		AUTO_WAITING_START,
		AUTO_WAITING_MODULES_READY,
		AUTO_WAITING_CAP,
		AUTO_DELIVERING_AND_PUNCHING_CAP,
		AUTO_SORTING_CAP,
		AUTO_WAITING_PICKUP_STATION_STOP,
		ERROR (*ERROR state*)
		);
	InternalType : 	STRUCT
		HeartBeatTimer : TON := (PT:=T#250MS);
		CommunicationTimeoutTimer : TON := (PT:=T#3S);
		PickingStationCommunicationOk : BOOL;
		OnPhaseStopRequest : BOOL;
		Error : BOOL;
		LastCapCounter : USINT;
	END_STRUCT;
END_TYPE
```

#### Variables.var - Local variables
```iecst
VAR
	MachineState : MachineStateType;
	Internal : InternalType;
	CommunicationInitialized : BOOL;
	CapWorkStopwatch : TON := (PT:=T#24d);
	CapsWorkingTimeHistory : ARRAY[0..STATS_HISTORY_MAX_INDEX] OF TIME;
	TotHistoryWorkedTime : TIME;
	Index : USINT;
END_VAR
```

#### Actions.st
```iecst
ACTION FeedbacksUpdateAction:

	gMainMachine.Feedbacks.WaitingInit := MachineState.ActualState = AUTO_WAITING_INIT;

	gMainMachine.Feedbacks.Initializing := MachineState.ActualState = AUTO_INITIALIZING;

	gMainMachine.Feedbacks.WaitingStart := MachineState.ActualState = AUTO_WAITING_START;

	gMainMachine.Feedbacks.WaitingModulesReady := MachineState.ActualState = AUTO_WAITING_MODULES_READY;

	gMainMachine.Feedbacks.PunchingCap := MachineState.ActualState = AUTO_DELIVERING_AND_PUNCHING_CAP AND gPuncher.Commands.Automatic.Start;

	gMainMachine.Feedbacks.WaitingCap := MachineState.ActualState = AUTO_WAITING_CAP;

	gMainMachine.Feedbacks.DeliveringCap := MachineState.ActualState = AUTO_DELIVERING_AND_PUNCHING_CAP;

	gMainMachine.Feedbacks.SortingCap := MachineState.ActualState = AUTO_SORTING_CAP;

	gMainMachine.Feedbacks.Error := MachineState.ActualState = ERROR;

	gMainMachine.Feedbacks.WaitModeSelection := MachineState.ActualState = WAITING_MODE_SELECTION;

	gMainMachine.Feedbacks.Stopping := gMainMachine.Feedbacks.Started AND Internal.OnPhaseStopRequest;

	gMainMachine.Feedbacks.ManualMode := (MachineState.ActualState = MANUAL);

	gMainMachine.Feedbacks.AutomaticMode := NOT gMainMachine.Feedbacks.ManualMode AND NOT gMainMachine.Feedbacks.WaitModeSelection AND NOT gMainMachine.Feedbacks.Error;

	IF gMainMachine.Commands.LinkMode THEN
		gMainMachine.Feedbacks.CapsOnConveyor := gConveyor.Feedbacks.CapsOnConveyor + gPickingStation.Outputs.CapsOnConveyor;
	ELSE
		gMainMachine.Feedbacks.CapsOnConveyor := gConveyor.Feedbacks.CapsOnConveyor;
	END_IF

	IF gMainMachine.Commands.Automatic.Init AND gMainMachine.Feedbacks.CapsOnConveyor > 0 THEN
		gMainMachine.Feedbacks.AskRemoveCaps := TRUE;
	ELSIF gMainMachine.Commands.Automatic.CapsRemoved THEN
		gMainMachine.Feedbacks.AskRemoveCaps := FALSE;
	END_IF

	// Started
	IF (MachineState.ActualState = AUTO_WAITING_MODULES_READY)
		OR (MachineState.ActualState = AUTO_WAITING_CAP)
		OR (MachineState.ActualState = AUTO_DELIVERING_AND_PUNCHING_CAP)
		OR (MachineState.ActualState = AUTO_SORTING_CAP) THEN

		gMainMachine.Feedbacks.Started := TRUE;
	ELSE
		gMainMachine.Feedbacks.Started := FALSE;
	END_IF

	IF NOT gMainMachine.Feedbacks.Started THEN
		gMainMachine.Feedbacks.NewCapOnWork := FALSE;
	END_IF

	IF NOT gMainMachine.Commands.Automatic.Init THEN
		gMainMachine.Feedbacks.InitDone := FALSE;
	END_IF
END_ACTION

ACTION MachineStateManagementAction:

    // Machine state timeout check
    MachineState.TimeoutTimer(IN := MachineState.TimeoutTimer.PT <> T#0S AND NOT MachineState.NewTriggerState);

	// Machine state change state logic
	MachineState.NewTriggerState := (MachineState.ActualState <> MachineState.NextState);
	IF MachineState.NewTriggerState THEN
		MachineState.OldState := MachineState.ActualState;
	END_IF
	MachineState.ActualState := MachineState.NextState;

END_ACTION

ACTION SetAlarmsAction:

	//Timeouts
	IF MachineState.TimeoutTimer.Q THEN

		// Throw here timeout alarms
		CASE MachineState.ActualState OF
			AUTO_INITIALIZING: MpAlarmXSet(gAlarmXCoreMpLink,'MainMachineInitializationTimeout'); // Edge alarm!
			AUTO_SORTING_CAP: MpAlarmXSet(gAlarmXCoreMpLink,'MainMachineCapMissing'); // Edge alarm!
			AUTO_DELIVERING_AND_PUNCHING_CAP: MpAlarmXSet(gAlarmXCoreMpLink,'MainMachineCapMissing'); // Edge alarm!
		END_CASE

		MachineState.NextState := ERROR;
	END_IF

	//MainMachineEmergencyCircuitInterrupted
	IF FALSE THEN
		MpAlarmXSet(gAlarmXCoreMpLink,'MainMachineEmergencyCircuitInterrupted'); // Persistent alarm
	ELSE
		MpAlarmXReset(gAlarmXCoreMpLink,'MainMachineEmergencyCircuitInterrupted'); // Persistent alarm
	END_IF

	//MainMachineCommunicationLost
	IF NOT Internal.PickingStationCommunicationOk AND gMainMachine.Commands.LinkMode THEN
		MpAlarmXSet(gAlarmXCoreMpLink,'MainMachineCommunicationLost');
	ELSE
		MpAlarmXReset(gAlarmXCoreMpLink,'MainMachineCommunicationLost');
	END_IF

	//MainMachinePickingStationInError
	IF gPickingStation.Outputs.Error AND gMainMachine.Commands.LinkMode AND NOT gMainMachine.Feedbacks.Error THEN
		MpAlarmXSet(gAlarmXCoreMpLink,'MainMachinePickingStationInError');
	END_IF

	//MainMachinePickingStationNotInLinkMode
	IF gMainMachine.Commands.LinkMode
		AND NOT gPickingStation.Outputs.LinkActive
		AND MachineState.ActualState <> MANUAL
		AND MachineState.ActualState <> ERROR
		AND MachineState.ActualState <> WAITING_MODE_SELECTION
		AND MachineState.ActualState <> AUTO_WAITING_INIT THEN
		MpAlarmXSet(gAlarmXCoreMpLink,'MainMachinePickingStationNotInLinkMode');
	ELSE
		MpAlarmXReset(gAlarmXCoreMpLink,'MainMachinePickingStationNotInLinkMode');
	END_IF

END_ACTION

ACTION PickingStationCommunication:

	// Send communication heart beat to picking station
	Internal.HeartBeatTimer(IN:=NOT Internal.HeartBeatTimer.Q);
	IF Internal.HeartBeatTimer.Q THEN
		gPickingStation.Inputs.HeartBeat := NOT gPickingStation.Inputs.HeartBeat;
	END_IF

	// Check communication heart beat from the slave
	IF EDGE(gPickingStation.Outputs.HeartBeat) THEN
		Internal.CommunicationTimeoutTimer.IN := FALSE;
		CommunicationInitialized := TRUE;
	ELSE
		Internal.CommunicationTimeoutTimer.IN := TRUE;
		IF Internal.CommunicationTimeoutTimer.Q THEN
			CommunicationInitialized := TRUE;
		END_IF

	END_IF

	Internal.CommunicationTimeoutTimer();

	Internal.PickingStationCommunicationOk := NOT Internal.CommunicationTimeoutTimer.Q AND CommunicationInitialized;
	gMainMachine.Feedbacks.LinkOk := Internal.PickingStationCommunicationOk;

END_ACTION

ACTION EnableModules:

	gColourSorter.Commands.Enable := TRUE;

	gConveyor.Commands.Enable := TRUE;

	gPuncher.Commands.Enable := TRUE;

END_ACTION

ACTION StopModules:

	gColourSorter.Commands.Manual.Enable := FALSE;
	gColourSorter.Commands.Automatic.Start := FALSE;
	gColourSorter.Commands.Automatic.Init := FALSE;
	gColourSorter.Commands.Reset := FALSE;

	gConveyor.Commands.Manual.Enable := FALSE;
	gConveyor.Commands.Automatic.Start := FALSE;
	gConveyor.Commands.Automatic.Init := FALSE;
	gConveyor.Commands.Reset := FALSE;
	gConveyor.Commands.Automatic.DecreaseCapCounter := FALSE;

	gPuncher.Commands.Manual.Enable := FALSE;
	gPuncher.Commands.Automatic.Start := FALSE;
	gPuncher.Commands.Automatic.Init := FALSE;
	gPuncher.Commands.Reset := FALSE;
	gPuncher.Commands.Automatic.PunchCap := FALSE;

	gPickingStation.Inputs.Start := FALSE;
	gPickingStation.Inputs.Init := FALSE;
	gPickingStation.Inputs.Reset := FALSE;

END_ACTION

ACTION ResetModulesManualCommands:

	memset(ADR(gColourSorter.Commands.Manual),0,SIZEOF(gColourSorter.Commands.Manual));
	memset(ADR(gPuncher.Commands.Manual),0,SIZEOF(gPuncher.Commands.Manual));
	memset(ADR(gConveyor.Commands.Manual),0,SIZEOF(gConveyor.Commands.Manual));

END_ACTION

ACTION InitModules:

	gColourSorter.Commands.Automatic.Init := TRUE;
	gConveyor.Commands.Automatic.Init := TRUE;
	gPuncher.Commands.Automatic.Init := TRUE;
	gPickingStation.Inputs.Init := TRUE;

END_ACTION

ACTION StartModules:

	gColourSorter.Commands.Automatic.Start := TRUE;
	gConveyor.Commands.Automatic.Start := TRUE;
	gPuncher.Commands.Automatic.Start := gMainMachine.Parameters.PuncherEnable;
	gPickingStation.Inputs.Start := TRUE;

END_ACTION

ACTION StatisticsAction:

	// Stats clear
	IF gMainMachine.Commands.ClearStats THEN
		memset(ADR(CapsWorkingTimeHistory),0,SIZEOF(CapsWorkingTimeHistory));
		gMainMachine.Statistics.CapsCounter := 0;
		gMainMachine.Feedbacks.ClearStatsDone := TRUE;
		CapWorkStopwatch.IN := FALSE;
	ELSE
		gMainMachine.Feedbacks.ClearStatsDone := FALSE;
	END_IF

	// Manage the stopwatch to measure the current cap working time
	IF EDGE(gMainMachine.Feedbacks.NewCapOnWork) THEN
		IF gMainMachine.Feedbacks.NewCapOnWork THEN
			gMainMachine.Statistics.CapsCounter := gMainMachine.Statistics.CapsCounter + 1;
			CapWorkStopwatch.IN := TRUE;
		ELSE
			CapWorkStopwatch.IN := FALSE;
			memmove(ADR(CapsWorkingTimeHistory[1]),ADR(CapsWorkingTimeHistory[0]),SIZEOF(CapsWorkingTimeHistory)-SIZEOF(CapsWorkingTimeHistory[0]));
			CapsWorkingTimeHistory[0] := CapWorkStopwatch.ET;
		END_IF
	END_IF

	CapWorkStopwatch();

	// Calc the total amount of time stored in the history array
	TotHistoryWorkedTime := T#0S;
	FOR Index:=0 TO STATS_HISTORY_MAX_INDEX DO
		IF CapsWorkingTimeHistory[Index]>T#0s THEN
			TotHistoryWorkedTime := TotHistoryWorkedTime + CapsWorkingTimeHistory[Index];
		ELSE
			EXIT;
		END_IF
	END_FOR

	gMainMachine.Statistics.CurrentCapWorkingTime := CapWorkStopwatch.ET;
	gMainMachine.Statistics.LastCapWorkingTime := CapsWorkingTimeHistory[0];
	gMainMachine.Statistics.AverageCapWorkingTime := UDINT_TO_TIME(TIME_TO_UDINT(TotHistoryWorkedTime)/MAX(1,Index));
END_ACTION

ACTION PickingStationAction:

	gPickingStation.Inputs.AutomaticMode := gMainMachine.Feedbacks.AutomaticMode;

	gPickingStation.Inputs.Error := gMainMachine.Feedbacks.Error;

	IF NOT gMainMachine.Commands.Automatic.Start THEN
		IF gMainMachine.Commands.LinkMode AND gPickingStation.Outputs.Started THEN
			gPickingStation.Inputs.Start := FALSE;
		END_IF
	END_IF
END_ACTION
```

### HMIGlobalTypes.typ
```iecst
TYPE
	HMIType : 	STRUCT  (*HMI Main type*)
		AutomaticPage : HMIAutomaticPageType;
		ManualPage : HMIManualPageType;
		HeaderContent : HMIHeaderContentType;
		RecipeContent : HMIRecipeContentType;
	END_STRUCT;
	HMIAutomaticPageType : 	STRUCT  (*HMI Interface Output type*)
		StartButtonEnable : BOOL;
		StartButton : BOOL;
		StopButtonVisibility : BOOL;
		InitButtonEnable : BOOL;
		InitButton : BOOL;
		ConveyorSpeed : REAL;
		ConveyorSpeedEnable : BOOL;
		AutoButtonEnable : BOOL;
		AutoButton : BOOL;
		LinkButtonEnable : BOOL;
		LinkButton : BOOL;
		ReadyToStartVisibility : BOOL;
		CurrentCapWorkingTime : UDINT;
		LastCapWorkedTime : UDINT;
		AvgCapWorkTime : UDINT;
		ClearStats : BOOL;
		PuncherIncludedCheckbox : BOOL;
		PuncherIncludedCheckboxEnable : BOOL;
		PuncherOffset : REAL;
		PuncherOffsetEnable : BOOL;
		CapsCounter : UDINT;
		StamperIncludedCheckbox : BOOL;
		StamperIncludedCheckboxEnable : BOOL;
		StamperOffset : REAL;
		StamperOffsetEnable : BOOL;
		RecipesEnable : BOOL;
		ShowLinkMsg : BOOL;
		AskRemoveCaps : BOOL;
		CapsRemoved : BOOL;
	END_STRUCT;
	HMIManualPageType : 	STRUCT  (*HMI Interface Output type*)
		ManualButtonEnable : BOOL;
		ManualButton : BOOL;
		StopperForwardButtonEnable : BOOL;
		StopperForwardButton : BOOL;
		Lane1ForwardButtonEnable : BOOL;
		Lane1ForwardButton : BOOL;
		Lane2ForwardButtonEnable : BOOL;
		Lane2ForwardButton : BOOL;
		ConveyorHomeButtonEnable : BOOL;
		ConveyorHomeButton : BOOL;
		ConveyorPowerButtonEnable : BOOL;
		ConveyorPowerButton : BOOL;
		ConveyorMoveButtonEnable : BOOL;
		ConveyorMoveButton : BOOL;
		ConveyorSpeed : REAL;
		ConveyorSpeedEnable : BOOL;
		ConveyorAxisHomed : BOOL;
		ConveyorAxisPowered : BOOL;
		PuncherHomeButtonEnable : BOOL;
		PuncherHomeButton : BOOL;
		PuncherPowerButtonEnable : BOOL;
		PuncherPowerButton : BOOL;
		PuncherMoveButtonEnable : BOOL;
		PuncherMoveButton : BOOL;
		PuncherSpeed : REAL;
		PuncherSpeedEnable : BOOL;
		PuncherAxisHomed : BOOL;
		PuncherAxisPowered : BOOL;
		PuncherForwardButtonEnable : BOOL;
		PuncherForwardButton : BOOL;
		PuncherPosition : LREAL;
		PuncherPositionEnable : BOOL;
		ColourSorterInterface : ColourSorterInterfaceType;
		ConveyorInterface : ConveyorInterfaceType;
		PuncherInterface : PuncherInterfaceType;
		ConveyorActSpeed : REAL;
		ConveyorActPosition : LREAL;
		PuncherActSpeed : REAL;
		PuncherActPosition : LREAL;
		ConveyorAcceleration : REAL;
		ConveyorAccelerationEnable : BOOL;
		PuncherAcceleration : REAL;
		PuncherAccelerationEnable : BOOL;
	END_STRUCT;
	HMIHeaderContentType : 	STRUCT  (*HMI Interface Output type*)
		SlaveConnectionOk : BOOL;
		PendingAlarms : STRING[3];
		StateManual : BOOL;
		StateWaitingInit : BOOL;
		StateInitializing : BOOL;
		StateWaitingStart : BOOL;
		StateWaitingModulesReady : BOOL;
		StateWaitingCap : BOOL;
		StatePunchingCap : BOOL;
		StateDeliveringCap : BOOL;
		StateError : BOOL;
		StateWaitModeSelection : BOOL;
		StateSortingCap : BOOL;
		ResetAlarms : BOOL;
		AlarmBlink : BOOL;
	END_STRUCT;
	HMIRecipeContentType : 	STRUCT  (*HMI Interface Output type*)
		EnableRecipesManagement : BOOL;
	END_STRUCT;
END_TYPE
```

### HMIGlobalVariables.var
```iecst
VAR
    gHMI : HMIType;
END_VAR
```

### Program Logical/Source/HMI/HMIProgram (IEC)

#### Main.st - Init, cyclic, exit code
```iecst
//******************************************************************************************************
// Program: 	HMIProgram
// Author: 		Andrea Pennisi
// Rev.: 		1.0.0
// Date:		5.12.2023
//
// Description:
// This module is used to manage the enables/visibility and value of the variable in the HMI
//******************************************************************************************************
PROGRAM _INIT
	SetInitialValuesAction;
END_PROGRAM

PROGRAM _CYCLIC

	HeaderContentAction;

	AutomaticPageAction;

	ManualPageAction;

	RecipeContentAction;

END_PROGRAM

PROGRAM _EXIT

END_PROGRAM
```

#### Variables.var - Local variables
```iecst
VAR
	AlarmBlinkTimer : TON;
END_VAR
```
